LIN {X 0,Y 411.207,Z 161.266,A -85,B 0,C 180,E1 -10595.783,E2 -10595.783} C_VEL
LIN {X 0,Y 411.182,Z 161.265,A -85,B 0,C 180,E1 -10598.965,E2 -10598.965} C_VEL
LIN {X 0,Y 411.239,Z 161.26,A -85,B 0,C 180,E1 -10602.084,E2 -10602.084} C_VEL
LIN {X 0,Y 411.248,Z 161.259,A -85,B 0,C 180,E1 -10605.147,E2 -10605.147} C_VEL
LIN {X 0,Y 411.282,Z 161.252,A -85,B 0,C 180,E1 -10608.167,E2 -10608.167} C_VEL
LIN {X 0,Y 411.428,Z 161.234,A -85,B 0,C 180,E1 -10612.185,E2 -10612.185} C_VEL
LIN {X 0,Y 411.463,Z 161.231,A -85,B 0,C 180,E1 -10614.118,E2 -10614.118} C_VEL
LIN {X 0,Y 411.499,Z 161.226,A -85,B 0,C 180,E1 -10618.042,E2 -10618.042} C_VEL
LIN {X 0,Y 411.626,Z 161.21,A -85,B 0,C 180,E1 -10620,E2 -10620} C_VEL
LIN {X 0,Y 411.439,Z 161.237,A -85,B 0,C 180,E1 -10622.937,E2 -10622.937} C_VEL
LIN {X 0,Y 411.445,Z 161.234,A -85,B 0,C 180,E1 -10626.867,E2 -10626.867} C_VEL
LIN {X 0,Y 411.294,Z 161.252,A -85,B 0,C 180,E1 -10629.839,E2 -10629.839} C_VEL
LIN {X 0,Y 411.299,Z 161.251,A -85,B 0,C 180,E1 -10633.11,E2 -10633.11} C_VEL
LIN {X 0,Y 411.243,Z 161.258,A -85,B 0,C 180,E1 -10636.889,E2 -10636.889} C_VEL
LIN {X 0,Y 411.241,Z 161.261,A -85,B 0,C 180,E1 -10639.986,E2 -10639.986} C_VEL
LIN {X 0,Y 411.192,Z 161.264,A -85,B 0,C 180,E1 -10643.148,E2 -10643.148} C_VEL
LIN {X 0,Y 411.182,Z 161.268,A -85,B 0,C 180,E1 -10646.385,E2 -10646.385} C_VEL
LIN {X 0,Y 411.185,Z 161.268,A -85,B 0,C 180,E1 -10649.714,E2 -10649.714} C_VEL
LIN {X 0,Y 411.194,Z 161.265,A -85,B 0,C 180,E1 -10653.157,E2 -10653.157} C_VEL
LIN {X 0,Y 411.184,Z 161.265,A -85,B 0,C 180,E1 -10656.554,E2 -10656.554} C_VEL
LIN {X 0,Y 411.207,Z 161.266,A -85,B 0,C 180,E1 -10659.73,E2 -10659.73} C_VEL
LIN {X 0,Y 411.167,Z 161.269,A -85,B 0,C 180,E1 -10663.134,E2 -10663.134} C_VEL
LIN {X 0,Y 411.164,Z 161.27,A -85,B 0,C 180,E1 -10665.882,E2 -10665.882} C_VEL
LIN {X 0,Y 411.155,Z 161.27,A -85,B 0,C 180,E1 -10668.773,E2 -10668.773} C_VEL
LIN {X 0,Y 411.183,Z 161.264,A -85,B 0,C 180,E1 -10672.028,E2 -10672.028} C_VEL
LIN {X 0,Y 411.198,Z 161.264,A -85,B 0,C 180,E1 -10675.668,E2 -10675.668} C_VEL
LIN {X 0,Y 411.194,Z 161.266,A -85,B 0,C 180,E1 -10679.155,E2 -10679.155} C_VEL
LIN {X 0,Y 411.254,Z 161.257,A -85,B 0,C 180,E1 -10682.524,E2 -10682.524} C_VEL
LIN {X 0,Y 411.212,Z 161.26,A -85,B 0,C 180,E1 -10685.786,E2 -10685.786} C_VEL
LIN {X 0,Y 411.193,Z 161.265,A -85,B 0,C 180,E1 -10688.968,E2 -10688.968} C_VEL
LIN {X 0,Y 411.251,Z 161.259,A -85,B 0,C 180,E1 -10692.087,E2 -10692.087} C_VEL
LIN {X 0,Y 411.257,Z 161.257,A -85,B 0,C 180,E1 -10695.149,E2 -10695.149} C_VEL
LIN {X 0,Y 411.282,Z 161.255,A -85,B 0,C 180,E1 -10698.169,E2 -10698.169} C_VEL
LIN {X 0,Y 411.482,Z 161.231,A -85,B 0,C 180,E1 -10702.148,E2 -10702.148} C_VEL
LIN {X 0,Y 411.476,Z 161.231,A -85,B 0,C 180,E1 -10704.12,E2 -10704.12} C_VEL
LIN {X 0,Y 411.512,Z 161.227,A -85,B 0,C 180,E1 -10708.044,E2 -10708.044} C_VEL
LIN {X 0,Y 411.379,Z 161.239,A -85,B 0,C 180,E1 -10710.98,E2 -10710.98} C_VEL
LIN {X 0,Y 411.452,Z 161.231,A -85,B 0,C 180,E1 -10712.939,E2 -10712.939} C_VEL
LIN {X 0,Y 411.464,Z 161.231,A -85,B 0,C 180,E1 -10716.868,E2 -10716.868} C_VEL
LIN {X 0,Y 411.357,Z 161.244,A -85,B 0,C 180,E1 -10718.847,E2 -10718.847} C_VEL
LIN {X 0,Y 411.287,Z 161.255,A -85,B 0,C 180,E1 -10721.834,E2 -10721.834} C_VEL
LIN {X 0,Y 411.26,Z 161.255,A -85,B 0,C 180,E1 -10724.854,E2 -10724.854} C_VEL
LIN {X 0,Y 411.243,Z 161.258,A -85,B 0,C 180,E1 -10727.609,E2 -10727.609} C_VEL
LIN {X 0,Y 410.583,Z 161.342,A -85,B 0,C 180,E1 -10728.427,E2 -10728.427} C_VEL
LIN {X 0,Y 407.695,Z 161.704,A -85,B 0,C 180,E1 -10729.755,E2 -10729.755} C_VEL
LIN {X 0,Y 405.251,Z 162.006,A -85,B 0,C 180,E1 -10730.827,E2 -10730.827} C_VEL
LIN {X 0,Y 404.215,Z 162.136,A -85,B 0,C 180,E1 -10731.657,E2 -10731.657} C_VEL
LIN {X 0,Y 404.138,Z 162.142,A -85,B 0,C 180,E1 -10731.938,E2 -10731.938} C_VEL
LIN {X 0,Y 404.156,Z 162.144,A -85,B 0,C 180,E1 -10735.278,E2 -10735.278} C_VEL
LIN {X 0,Y 404.156,Z 162.143,A -85,B 0,C 180,E1 -10739.139,E2 -10739.139} C_VEL
LIN {X 0,Y 404.146,Z 162.144,A -85,B 0,C 180,E1 -10742.623,E2 -10742.623} C_VEL
LIN {X 0,Y 404.184,Z 162.14,A -85,B 0,C 180,E1 -10745.19,E2 -10745.19} C_VEL
LIN {X 0,Y 404.137,Z 162.147,A -85,B 0,C 180,E1 -10748.76,E2 -10748.76} C_VEL
LIN {X 0,Y 404.113,Z 162.145,A -85,B 0,C 180,E1 -10751.598,E2 -10751.598} C_VEL
LIN {X 0,Y 404.149,Z 162.143,A -85,B 0,C 180,E1 -10754.523,E2 -10754.523} C_VEL
LIN {X 0,Y 404.142,Z 162.142,A -85,B 0,C 180,E1 -10757.296,E2 -10757.296} C_VEL
LIN {X 0,Y 404.137,Z 162.144,A -85,B 0,C 180,E1 -10759.952,E2 -10759.952} C_VEL
LIN {X 0,Y 404.137,Z 162.142,A -85,B 0,C 180,E1 -10763.127,E2 -10763.127} C_VEL
LIN {X 0,Y 404.212,Z 162.136,A -85,B 0,C 180,E1 -10766.573,E2 -10766.573} C_VEL
LIN {X 0,Y 404.224,Z 162.166,A -85,B 0,C 180,E1 -10766.845,E2 -10766.845} C_VEL
LIN {X 0,Y 405.07,Z 167.315,A -85,B 0,C 180,E1 -10769.214,E2 -10769.214} C_VEL
LIN {X 0,Y 404.937,Z 172.513,A -85,B 0,C 180,E1 -10771.492,E2 -10771.492} C_VEL
LIN {X 0,Y 404.575,Z 179.708,A -85,B 0,C 180,E1 -10774.599,E2 -10774.599} C_VEL
LIN {X 0,Y 404.159,Z 187.845,A -85,B 0,C 180,E1 -10778.046,E2 -10778.046} C_VEL
LIN {X 0,Y 403.86,Z 195.462,A -85,B 0,C 180,E1 -10781.22,E2 -10781.22} C_VEL
LIN {X 0,Y 403.622,Z 203.044,A -85,B 0,C 180,E1 -10784.342,E2 -10784.342} C_VEL
LIN {X 0,Y 403.35,Z 211.861,A -85,B 0,C 180,E1 -10787.931,E2 -10787.931} C_VEL
LIN {X 0,Y 403.222,Z 215.611,A -85,B 0,C 180,E1 -10789.423,E2 -10789.423} C_VEL
LIN {X 0,Y 404.314,Z 226.159,A -85,B 0,C 180,E1 -10789.99,E2 -10789.99} C_VEL
LIN {X 0,Y 404.795,Z 233.544,A -85,B 0,C 180,E1 -10790.506,E2 -10790.506} C_VEL
LIN {X 0,Y 404.342,Z 243.511,A -85,B 0,C 180,E1 -10791.378,E2 -10791.378} C_VEL
LIN {X 0,Y 404.028,Z 251.821,A -85,B 0,C 180,E1 -10792.322,E2 -10792.322} C_VEL
LIN {X 0,Y 403.71,Z 259.93,A -85,B 0,C 180,E1 -10793.503,E2 -10793.503} C_VEL
LIN {X 0,Y 403.453,Z 266.509,A -85,B 0,C 180,E1 -10794.753,E2 -10794.753} C_VEL
LIN {X 0,Y 403.306,Z 271.492,A -85,B 0,C 180,E1 -10796.003,E2 -10796.003} C_VEL
LIN {X 0,Y 403.07,Z 275.759,A -85,B 0,C 180,E1 -10797.502,E2 -10797.502} C_VEL
LIN {X 0,Y 402.968,Z 278.356,A -85,B 0,C 180,E1 -10799.001,E2 -10799.001} C_VEL
LIN {X 0,Y 402.972,Z 279.231,A -85,B 0,C 180,E1 -10800,E2 -10800} C_VEL
LIN {X 0,Y 403.052,Z 279.432,A -85,B 0,C 180,E1 -10800.999,E2 -10800.999} C_VEL
LIN {X 0,Y 403.192,Z 278.964,A -85,B 0,C 180,E1 -10801.998,E2 -10801.998} C_VEL
LIN {X 0,Y 403.41,Z 277.828,A -85,B 0,C 180,E1 -10802.996,E2 -10802.996} C_VEL
LIN {X 0,Y 403.747,Z 274.846,A -85,B 0,C 180,E1 -10804.493,E2 -10804.493} C_VEL
LIN {X 0,Y 404.065,Z 270.202,A -85,B 0,C 180,E1 -10805.99,E2 -10805.99} C_VEL
LIN {X 0,Y 404.434,Z 264.853,A -85,B 0,C 180,E1 -10807.238,E2 -10807.238} C_VEL
LIN {X 0,Y 405.159,Z 257.556,A -85,B 0,C 180,E1 -10808.529,E2 -10808.529} C_VEL
LIN {X 0,Y 405.943,Z 248.74,A -85,B 0,C 180,E1 -10809.718,E2 -10809.718} C_VEL
LIN {X 0,Y 406.748,Z 239.232,A -85,B 0,C 180,E1 -10810.705,E2 -10810.705} C_VEL
LIN {X 0,Y 406.752,Z 233.542,A -85,B 0,C 180,E1 -10811.209,E2 -10811.209} C_VEL
LIN {X 0,Y 405.297,Z 223.531,A -85,B 0,C 180,E1 -10812.01,E2 -10812.01} C_VEL
LIN {X 0,Y 403.844,Z 216.665,A -85,B 0,C 180,E1 -10812.507,E2 -10812.507} C_VEL
LIN {X 0,Y 404.246,Z 209.533,A -85,B 0,C 180,E1 -10815.633,E2 -10815.633} C_VEL
LIN {X 0,Y 404.678,Z 202.657,A -85,B 0,C 180,E1 -10818.741,E2 -10818.741} C_VEL
LIN {X 0,Y 405.281,Z 194.834,A -85,B 0,C 180,E1 -10822.427,E2 -10822.427} C_VEL
LIN {X 0,Y 406.002,Z 188.022,A -85,B 0,C 180,E1 -10825.822,E2 -10825.822} C_VEL
LIN {X 0,Y 406.894,Z 182.208,A -85,B 0,C 180,E1 -10828.923,E2 -10828.923} C_VEL
LIN {X 0,Y 407.201,Z 178.392,A -85,B 0,C 180,E1 -10831.184,E2 -10831.184} C_VEL
LIN {X 0,Y 406.895,Z 175.006,A -85,B 0,C 180,E1 -10833.554,E2 -10833.554} C_VEL
LIN {X 0,Y 406.335,Z 172.065,A -85,B 0,C 180,E1 -10836.02,E2 -10836.02} C_VEL
LIN {X 0,Y 405.886,Z 169.428,A -85,B 0,C 180,E1 -10838.812,E2 -10838.812} C_VEL
LIN {X 0,Y 405.452,Z 167.68,A -85,B 0,C 180,E1 -10841.809,E2 -10841.809} C_VEL
LIN {X 0,Y 405.365,Z 167.011,A -85,B 0,C 180,E1 -10844.696,E2 -10844.696} C_VEL
LIN {X 0,Y 405.483,Z 167.548,A -85,B 0,C 180,E1 -10847.469,E2 -10847.469} C_VEL
LIN {X 0,Y 405.882,Z 169.048,A -85,B 0,C 180,E1 -10850.157,E2 -10850.157} C_VEL
LIN {X 0,Y 406.461,Z 171.553,A -85,B 0,C 180,E1 -10852.757,E2 -10852.757} C_VEL
LIN {X 0,Y 407.472,Z 175.865,A -85,B 0,C 180,E1 -10855.884,E2 -10855.884} C_VEL
LIN {X 0,Y 408.63,Z 181.39,A -85,B 0,C 180,E1 -10858.936,E2 -10858.936} C_VEL
LIN {X 0,Y 409.421,Z 186.484,A -85,B 0,C 180,E1 -10861.271,E2 -10861.271} C_VEL
LIN {X 0,Y 408.85,Z 190.802,A -85,B 0,C 180,E1 -10862.9,E2 -10862.9} C_VEL
LIN {X 0,Y 407.122,Z 200.495,A -85,B 0,C 180,E1 -10866.195,E2 -10866.195} C_VEL
LIN {X 0,Y 405.713,Z 211.784,A -85,B 0,C 180,E1 -10869.728,E2 -10869.728} C_VEL
LIN {X 0,Y 404.899,Z 220.511,A -85,B 0,C 180,E1 -10872.295,E2 -10872.295} C_VEL
LIN {X 0,Y 407.213,Z 233.303,A -85,B 0,C 180,E1 -10872.87,E2 -10872.87} C_VEL
LIN {X 0,Y 407.871,Z 244.837,A -85,B 0,C 180,E1 -10873.481,E2 -10873.481} C_VEL
LIN {X 0,Y 407.187,Z 256.391,A -85,B 0,C 180,E1 -10874.225,E2 -10874.225} C_VEL
LIN {X 0,Y 406.24,Z 268.36,A -85,B 0,C 180,E1 -10875.215,E2 -10875.215} C_VEL
LIN {X 0,Y 405.341,Z 278.907,A -85,B 0,C 180,E1 -10876.327,E2 -10876.327} C_VEL
LIN {X 0,Y 404.683,Z 289.375,A -85,B 0,C 180,E1 -10877.715,E2 -10877.715} C_VEL
LIN {X 0,Y 403.867,Z 298.395,A -85,B 0,C 180,E1 -10879.217,E2 -10879.217} C_VEL
LIN {X 0,Y 403.427,Z 305.665,A -85,B 0,C 180,E1 -10880.725,E2 -10880.725} C_VEL
LIN {X 0,Y 403.192,Z 310.558,A -85,B 0,C 180,E1 -10881.983,E2 -10881.983} C_VEL
LIN {X 0,Y 403.004,Z 315.426,A -85,B 0,C 180,E1 -10883.54,E2 -10883.54} C_VEL
LIN {X 0,Y 402.961,Z 318.87,A -85,B 0,C 180,E1 -10884.996,E2 -10884.996} C_VEL
LIN {X 0,Y 402.885,Z 320.644,A -85,B 0,C 180,E1 -10885.997,E2 -10885.997} C_VEL
LIN {X 0,Y 402.918,Z 322.001,A -85,B 0,C 180,E1 -10886.999,E2 -10886.999} C_VEL
LIN {X 0,Y 402.969,Z 322.941,A -85,B 0,C 180,E1 -10888,E2 -10888} C_VEL
LIN {X 0,Y 402.929,Z 323.408,A -85,B 0,C 180,E1 -10888.999,E2 -10888.999} C_VEL
LIN {X 0,Y 402.958,Z 323.469,A -85,B 0,C 180,E1 -10889.998,E2 -10889.998} C_VEL
LIN {X 0,Y 402.962,Z 323.121,A -85,B 0,C 180,E1 -10890.998,E2 -10890.998} C_VEL
LIN {X 0,Y 402.989,Z 322.303,A -85,B 0,C 180,E1 -10891.997,E2 -10891.997} C_VEL
LIN {X 0,Y 403.004,Z 321.057,A -85,B 0,C 180,E1 -10892.997,E2 -10892.997} C_VEL
LIN {X 0,Y 402.95,Z 318.326,A -85,B 0,C 180,E1 -10894.5,E2 -10894.5} C_VEL
LIN {X 0,Y 402.986,Z 314.496,A -85,B 0,C 180,E1 -10896.005,E2 -10896.005} C_VEL
LIN {X 0,Y 403.126,Z 309.461,A -85,B 0,C 180,E1 -10897.511,E2 -10897.511} C_VEL
LIN {X 0,Y 403.313,Z 302.989,A -85,B 0,C 180,E1 -10899.021,E2 -10899.021} C_VEL
LIN {X 0,Y 403.674,Z 294.844,A -85,B 0,C 180,E1 -10900.531,E2 -10900.531} C_VEL
LIN {X 0,Y 404.185,Z 286.47,A -85,B 0,C 180,E1 -10901.787,E2 -10901.787} C_VEL
LIN {X 0,Y 404.704,Z 277.19,A -85,B 0,C 180,E1 -10902.918,E2 -10902.918} C_VEL
LIN {X 0,Y 405.199,Z 265.616,A -85,B 0,C 180,E1 -10904.051,E2 -10904.051} C_VEL
LIN {X 0,Y 405.85,Z 254.099,A -85,B 0,C 180,E1 -10904.925,E2 -10904.925} C_VEL
LIN {X 0,Y 406.283,Z 242.176,A -85,B 0,C 180,E1 -10905.615,E2 -10905.615} C_VEL
LIN {X 0,Y 405.168,Z 230.504,A -85,B 0,C 180,E1 -10906.139,E2 -10906.139} C_VEL
LIN {X 0,Y 404.151,Z 220.278,A -85,B 0,C 180,E1 -10906.49,E2 -10906.49} C_VEL
LIN {X 0,Y 405.068,Z 206.335,A -85,B 0,C 180,E1 -10910.302,E2 -10910.302} C_VEL
LIN {X 0,Y 406.165,Z 193.07,A -85,B 0,C 180,E1 -10913.991,E2 -10913.991} C_VEL
LIN {X 0,Y 407.256,Z 181.733,A -85,B 0,C 180,E1 -10917.211,E2 -10917.211} C_VEL
LIN {X 0,Y 407.239,Z 177.881,A -85,B 0,C 180,E1 -10918.34,E2 -10918.34} C_VEL
LIN {X 0,Y 405.33,Z 168.24,A -85,B 0,C 180,E1 -10921.341,E2 -10921.341} C_VEL
LIN {X 0,Y 404.145,Z 162.145,A -85,B 0,C 180,E1 -10923.327,E2 -10923.327} C_VEL
LIN {X 0,Y 404.137,Z 162.147,A -85,B 0,C 180,E1 -10926.244,E2 -10926.244} C_VEL
LIN {X 0,Y 404.143,Z 162.145,A -85,B 0,C 180,E1 -10928.756,E2 -10928.756} C_VEL
LIN {X 0,Y 404.11,Z 162.144,A -85,B 0,C 180,E1 -10931.597,E2 -10931.597} C_VEL
LIN {X 0,Y 404.144,Z 162.145,A -85,B 0,C 180,E1 -10934.522,E2 -10934.522} C_VEL
LIN {X 0,Y 404.201,Z 162.135,A -85,B 0,C 180,E1 -10937.304,E2 -10937.304} C_VEL
LIN {X 0,Y 404.159,Z 162.142,A -85,B 0,C 180,E1 -10939.954,E2 -10939.954} C_VEL
LIN {X 0,Y 404.126,Z 162.143,A -85,B 0,C 180,E1 -10943.124,E2 -10943.124} C_VEL
LIN {X 0,Y 404.133,Z 162.146,A -85,B 0,C 180,E1 -10946.186,E2 -10946.186} C_VEL
LIN {X 0,Y 404.142,Z 162.146,A -85,B 0,C 180,E1 -10949.714,E2 -10949.714} C_VEL
LIN {X 0,Y 404.182,Z 162.138,A -85,B 0,C 180,E1 -10953.122,E2 -10953.122} C_VEL
LIN {X 0,Y 404.161,Z 162.14,A -85,B 0,C 180,E1 -10955.333,E2 -10955.333} C_VEL
LIN {X 0,Y 404.124,Z 162.144,A -85,B 0,C 180,E1 -10958.58,E2 -10958.58} C_VEL
LIN {X 0,Y 404.196,Z 162.137,A -85,B 0,C 180,E1 -10961.761,E2 -10961.761} C_VEL
LIN {X 0,Y 404.193,Z 162.137,A -85,B 0,C 180,E1 -10964.881,E2 -10964.881} C_VEL
LIN {X 0,Y 404.253,Z 162.129,A -85,B 0,C 180,E1 -10967.958,E2 -10967.958} C_VEL
LIN {X 0,Y 404.391,Z 162.111,A -85,B 0,C 180,E1 -10972.127,E2 -10972.127} C_VEL
LIN {X 0,Y 404.411,Z 162.109,A -85,B 0,C 180,E1 -10974.015,E2 -10974.015} C_VEL
LIN {X 0,Y 404.468,Z 162.102,A -85,B 0,C 180,E1 -10978.008,E2 -10978.008} C_VEL
LIN {X 0,Y 404.595,Z 162.085,A -85,B 0,C 180,E1 -10980,E2 -10980} C_VEL
LIN {X 0,Y 404.397,Z 162.114,A -85,B 0,C 180,E1 -10982.989,E2 -10982.989} C_VEL
LIN {X 0,Y 404.396,Z 162.112,A -85,B 0,C 180,E1 -10986.987,E2 -10986.987} C_VEL
LIN {X 0,Y 404.257,Z 162.129,A -85,B 0,C 180,E1 -10990.012,E2 -10990.012} C_VEL
LIN {X 0,Y 404.252,Z 162.128,A -85,B 0,C 180,E1 -10993.212,E2 -10993.212} C_VEL
LIN {X 0,Y 404.201,Z 162.135,A -85,B 0,C 180,E1 -10997.008,E2 -10997.008} C_VEL
LIN {X 0,Y 404.187,Z 162.139,A -85,B 0,C 180,E1 -11000.35,E2 -11000.35} C_VEL
LIN {X 0,Y 404.155,Z 162.142,A -85,B 0,C 180,E1 -11003.575,E2 -11003.575} C_VEL
LIN {X 0,Y 404.121,Z 162.144,A -85,B 0,C 180,E1 -11006.882,E2 -11006.882} C_VEL
LIN {X 0,Y 404.131,Z 162.145,A -85,B 0,C 180,E1 -11010.286,E2 -11010.286} C_VEL
LIN {X 0,Y 404.133,Z 162.146,A -85,B 0,C 180,E1 -11013.813,E2 -11013.813} C_VEL
LIN {X 0,Y 404.128,Z 162.144,A -85,B 0,C 180,E1 -11016.877,E2 -11016.877} C_VEL
LIN {X 0,Y 404.137,Z 162.143,A -85,B 0,C 180,E1 -11020.082,E2 -11020.082} C_VEL
LIN {X 0,Y 404.146,Z 162.143,A -85,B 0,C 180,E1 -11023.086,E2 -11023.086} C_VEL
LIN {X 0,Y 404.143,Z 162.144,A -85,B 0,C 180,E1 -11025.928,E2 -11025.928} C_VEL
LIN {X 0,Y 404.11,Z 162.147,A -85,B 0,C 180,E1 -11028.637,E2 -11028.637} C_VEL
LIN {X 0,Y 404.141,Z 162.145,A -85,B 0,C 180,E1 -11031.495,E2 -11031.495} C_VEL
LIN {X 0,Y 404.177,Z 162.142,A -85,B 0,C 180,E1 -11034.986,E2 -11034.986} C_VEL
LIN {X 0,Y 404.141,Z 162.144,A -85,B 0,C 180,E1 -11038.556,E2 -11038.556} C_VEL
LIN {X 0,Y 404.192,Z 162.136,A -85,B 0,C 180,E1 -11042.002,E2 -11042.002} C_VEL
LIN {X 0,Y 404.168,Z 162.139,A -85,B 0,C 180,E1 -11045.336,E2 -11045.336} C_VEL
LIN {X 0,Y 404.156,Z 162.144,A -85,B 0,C 180,E1 -11048.584,E2 -11048.584} C_VEL
LIN {X 0,Y 404.208,Z 162.134,A -85,B 0,C 180,E1 -11051.764,E2 -11051.764} C_VEL
LIN {X 0,Y 404.203,Z 162.137,A -85,B 0,C 180,E1 -11054.884,E2 -11054.884} C_VEL
LIN {X 0,Y 404.254,Z 162.129,A -85,B 0,C 180,E1 -11057.96,E2 -11057.96} C_VEL
LIN {X 0,Y 404.434,Z 162.109,A -85,B 0,C 180,E1 -11062.101,E2 -11062.101} C_VEL
LIN {X 0,Y 404.425,Z 162.11,A -85,B 0,C 180,E1 -11064.017,E2 -11064.017} C_VEL
LIN {X 0,Y 404.481,Z 162.102,A -85,B 0,C 180,E1 -11068.01,E2 -11068.01} C_VEL
LIN {X 0,Y 404.349,Z 162.115,A -85,B 0,C 180,E1 -11070.997,E2 -11070.997} C_VEL
LIN {X 0,Y 404.41,Z 162.108,A -85,B 0,C 180,E1 -11072.99,E2 -11072.99} C_VEL
LIN {X 0,Y 404.415,Z 162.109,A -85,B 0,C 180,E1 -11076.989,E2 -11076.989} C_VEL
LIN {X 0,Y 404.26,Z 162.13,A -85,B 0,C 180,E1 -11080.013,E2 -11080.013} C_VEL
LIN {X 0,Y 404.27,Z 162.127,A -85,B 0,C 180,E1 -11083.213,E2 -11083.213} C_VEL
LIN {X 0,Y 404.22,Z 162.135,A -85,B 0,C 180,E1 -11087.008,E2 -11087.008} C_VEL
LIN {X 0,Y 404.168,Z 162.139,A -85,B 0,C 180,E1 -11090.353,E2 -11090.353} C_VEL
LIN {X 0,Y 404.138,Z 162.142,A -85,B 0,C 180,E1 -11091.938,E2 -11091.938} C_VEL
LIN {X 0,Y 403.497,Z 162.224,A -85,B 0,C 180,E1 -11092.77,E2 -11092.77} C_VEL
LIN {X 0,Y 400.665,Z 162.576,A -85,B 0,C 180,E1 -11094.121,E2 -11094.121} C_VEL
LIN {X 0,Y 398.238,Z 162.882,A -85,B 0,C 180,E1 -11095.213,E2 -11095.213} C_VEL
LIN {X 0,Y 397.173,Z 163.01,A -85,B 0,C 180,E1 -11096.056,E2 -11096.056} C_VEL
LIN {X 0,Y 397.074,Z 163.02,A -85,B 0,C 180,E1 -11096.342,E2 -11096.342} C_VEL
LIN {X 0,Y 397.104,Z 163.019,A -85,B 0,C 180,E1 -11099.864,E2 -11099.864} C_VEL
LIN {X 0,Y 397.123,Z 163.017,A -85,B 0,C 180,E1 -11103.719,E2 -11103.719} C_VEL
LIN {X 0,Y 397.093,Z 163.021,A -85,B 0,C 180,E1 -11107.209,E2 -11107.209} C_VEL
LIN {X 0,Y 397.06,Z 163.027,A -85,B 0,C 180,E1 -11110.438,E2 -11110.438} C_VEL
LIN {X 0,Y 397.103,Z 163.019,A -85,B 0,C 180,E1 -11113.65,E2 -11113.65} C_VEL
LIN {X 0,Y 397.107,Z 163.021,A -85,B 0,C 180,E1 -11116.522,E2 -11116.522} C_VEL
LIN {X 0,Y 397.107,Z 163.018,A -85,B 0,C 180,E1 -11119.555,E2 -11119.555} C_VEL
LIN {X 0,Y 397.099,Z 163.019,A -85,B 0,C 180,E1 -11123.005,E2 -11123.005} C_VEL
LIN {X 0,Y 397.179,Z 163.072,A -85,B 0,C 180,E1 -11126.733,E2 -11126.733} C_VEL
LIN {X 0,Y 398.056,Z 168.37,A -85,B 0,C 180,E1 -11129.202,E2 -11129.202} C_VEL
LIN {X 0,Y 397.847,Z 174.757,A -85,B 0,C 180,E1 -11132.039,E2 -11132.039} C_VEL
LIN {X 0,Y 397.474,Z 181.305,A -85,B 0,C 180,E1 -11134.89,E2 -11134.89} C_VEL
LIN {X 0,Y 397.066,Z 190.251,A -85,B 0,C 180,E1 -11138.725,E2 -11138.725} C_VEL
LIN {X 0,Y 396.694,Z 199.128,A -85,B 0,C 180,E1 -11142.472,E2 -11142.472} C_VEL
LIN {X 0,Y 396.395,Z 207.989,A -85,B 0,C 180,E1 -11146.152,E2 -11146.152} C_VEL
LIN {X 0,Y 396.182,Z 215.595,A -85,B 0,C 180,E1 -11149.265,E2 -11149.265} C_VEL
LIN {X 0,Y 397.347,Z 227.437,A -85,B 0,C 180,E1 -11149.941,E2 -11149.941} C_VEL
LIN {X 0,Y 397.711,Z 234.605,A -85,B 0,C 180,E1 -11150.464,E2 -11150.464} C_VEL
LIN {X 0,Y 397.252,Z 244.375,A -85,B 0,C 180,E1 -11151.351,E2 -11151.351} C_VEL
LIN {X 0,Y 396.901,Z 253.364,A -85,B 0,C 180,E1 -11152.42,E2 -11152.42} C_VEL
LIN {X 0,Y 396.646,Z 260.068,A -85,B 0,C 180,E1 -11153.432,E2 -11153.432} C_VEL
LIN {X 0,Y 396.397,Z 266.487,A -85,B 0,C 180,E1 -11154.659,E2 -11154.659} C_VEL
LIN {X 0,Y 396.216,Z 271.57,A -85,B 0,C 180,E1 -11155.931,E2 -11155.931} C_VEL
LIN {X 0,Y 396.004,Z 275.949,A -85,B 0,C 180,E1 -11157.457,E2 -11157.457} C_VEL
LIN {X 0,Y 395.893,Z 278.654,A -85,B 0,C 180,E1 -11158.983,E2 -11158.983} C_VEL
LIN {X 0,Y 395.893,Z 279.596,A -85,B 0,C 180,E1 -11160,E2 -11160} C_VEL
LIN {X 0,Y 395.973,Z 279.868,A -85,B 0,C 180,E1 -11161.017,E2 -11161.017} C_VEL
LIN {X 0,Y 396.118,Z 279.475,A -85,B 0,C 180,E1 -11162.034,E2 -11162.034} C_VEL
LIN {X 0,Y 396.346,Z 278.414,A -85,B 0,C 180,E1 -11163.049,E2 -11163.049} C_VEL
LIN {X 0,Y 396.719,Z 275.551,A -85,B 0,C 180,E1 -11164.573,E2 -11164.573} C_VEL
LIN {X 0,Y 397.06,Z 271.053,A -85,B 0,C 180,E1 -11166.096,E2 -11166.096} C_VEL
LIN {X 0,Y 397.439,Z 266.033,A -85,B 0,C 180,E1 -11167.33,E2 -11167.33} C_VEL
LIN {X 0,Y 398.202,Z 259.079,A -85,B 0,C 180,E1 -11168.629,E2 -11168.629} C_VEL
LIN {X 0,Y 399.072,Z 250.28,A -85,B 0,C 180,E1 -11169.887,E2 -11169.887} C_VEL
LIN {X 0,Y 399.921,Z 241.18,A -85,B 0,C 180,E1 -11170.89,E2 -11170.89} C_VEL
LIN {X 0,Y 400.101,Z 235.734,A -85,B 0,C 180,E1 -11171.397,E2 -11171.397} C_VEL
LIN {X 0,Y 398.891,Z 226.392,A -85,B 0,C 180,E1 -11172.206,E2 -11172.206} C_VEL
LIN {X 0,Y 396.89,Z 216.809,A -85,B 0,C 180,E1 -11172.936,E2 -11172.936} C_VEL
LIN {X 0,Y 397.344,Z 209.011,A -85,B 0,C 180,E1 -11176.439,E2 -11176.439} C_VEL
LIN {X 0,Y 397.828,Z 202.204,A -85,B 0,C 180,E1 -11179.612,E2 -11179.612} C_VEL
LIN {X 0,Y 398.421,Z 195.601,A -85,B 0,C 180,E1 -11182.835,E2 -11182.835} C_VEL
LIN {X 0,Y 399.182,Z 189.217,A -85,B 0,C 180,E1 -11186.114,E2 -11186.114} C_VEL
LIN {X 0,Y 399.897,Z 184.831,A -85,B 0,C 180,E1 -11188.509,E2 -11188.509} C_VEL
LIN {X 0,Y 400.346,Z 181.227,A -85,B 0,C 180,E1 -11190.661,E2 -11190.661} C_VEL
LIN {X 0,Y 400.205,Z 177.886,A -85,B 0,C 180,E1 -11192.983,E2 -11192.983} C_VEL
LIN {X 0,Y 399.628,Z 174.35,A -85,B 0,C 180,E1 -11196.003,E2 -11196.003} C_VEL
LIN {X 0,Y 399.126,Z 171.446,A -85,B 0,C 180,E1 -11199.339,E2 -11199.339} C_VEL
LIN {X 0,Y 398.778,Z 169.993,A -85,B 0,C 180,E1 -11202.25,E2 -11202.25} C_VEL
LIN {X 0,Y 398.752,Z 169.62,A -85,B 0,C 180,E1 -11205.169,E2 -11205.169} C_VEL
LIN {X 0,Y 398.911,Z 170.331,A -85,B 0,C 180,E1 -11207.971,E2 -11207.971} C_VEL
LIN {X 0,Y 399.385,Z 172.082,A -85,B 0,C 180,E1 -11210.739,E2 -11210.739} C_VEL
LIN {X 0,Y 400.151,Z 175.491,A -85,B 0,C 180,E1 -11213.893,E2 -11213.893} C_VEL
LIN {X 0,Y 401.005,Z 179.27,A -85,B 0,C 180,E1 -11216.49,E2 -11216.49} C_VEL
LIN {X 0,Y 401.926,Z 183.711,A -85,B 0,C 180,E1 -11218.96,E2 -11218.96} C_VEL
LIN {X 0,Y 402.606,Z 188.858,A -85,B 0,C 180,E1 -11221.345,E2 -11221.345} C_VEL
LIN {X 0,Y 401.826,Z 193.533,A -85,B 0,C 180,E1 -11223.126,E2 -11223.126} C_VEL
LIN {X 0,Y 400.175,Z 202.295,A -85,B 0,C 180,E1 -11226.174,E2 -11226.174} C_VEL
LIN {X 0,Y 398.863,Z 212.184,A -85,B 0,C 180,E1 -11229.364,E2 -11229.364} C_VEL
LIN {X 0,Y 398.027,Z 220.376,A -85,B 0,C 180,E1 -11231.857,E2 -11231.857} C_VEL
LIN {X 0,Y 400.43,Z 233.45,A -85,B 0,C 180,E1 -11232.494,E2 -11232.494} C_VEL
LIN {X 0,Y 401.188,Z 243.95,A -85,B 0,C 180,E1 -11233.077,E2 -11233.077} C_VEL
LIN {X 0,Y 400.516,Z 255.473,A -85,B 0,C 180,E1 -11233.824,E2 -11233.824} C_VEL
LIN {X 0,Y 399.55,Z 267.51,A -85,B 0,C 180,E1 -11234.831,E2 -11234.831} C_VEL
LIN {X 0,Y 398.58,Z 277.977,A -85,B 0,C 180,E1 -11235.94,E2 -11235.94} C_VEL
LIN {X 0,Y 397.943,Z 286.02,A -85,B 0,C 180,E1 -11236.985,E2 -11236.985} C_VEL
LIN {X 0,Y 397.293,Z 294.184,A -85,B 0,C 180,E1 -11238.261,E2 -11238.261} C_VEL
LIN {X 0,Y 396.653,Z 302.202,A -85,B 0,C 180,E1 -11239.793,E2 -11239.793} C_VEL
LIN {X 0,Y 396.215,Z 308.577,A -85,B 0,C 180,E1 -11241.327,E2 -11241.327} C_VEL
LIN {X 0,Y 396.002,Z 313.635,A -85,B 0,C 180,E1 -11242.862,E2 -11242.862} C_VEL
LIN {X 0,Y 395.832,Z 317.074,A -85,B 0,C 180,E1 -11244.187,E2 -11244.187} C_VEL
LIN {X 0,Y 395.806,Z 320.34,A -85,B 0,C 180,E1 -11245.926,E2 -11245.926} C_VEL
LIN {X 0,Y 395.817,Z 321.672,A -85,B 0,C 180,E1 -11246.945,E2 -11246.945} C_VEL
LIN {X 0,Y 395.898,Z 322.567,A -85,B 0,C 180,E1 -11247.964,E2 -11247.964} C_VEL
LIN {X 0,Y 395.855,Z 323.004,A -85,B 0,C 180,E1 -11248.981,E2 -11248.981} C_VEL
LIN {X 0,Y 395.88,Z 323.039,A -85,B 0,C 180,E1 -11249.998,E2 -11249.998} C_VEL
LIN {X 0,Y 395.886,Z 322.648,A -85,B 0,C 180,E1 -11251.016,E2 -11251.016} C_VEL
LIN {X 0,Y 395.92,Z 321.791,A -85,B 0,C 180,E1 -11252.033,E2 -11252.033} C_VEL
LIN {X 0,Y 395.906,Z 320.514,A -85,B 0,C 180,E1 -11253.051,E2 -11253.051} C_VEL
LIN {X 0,Y 395.884,Z 317.722,A -85,B 0,C 180,E1 -11254.58,E2 -11254.58} C_VEL
LIN {X 0,Y 395.953,Z 313.287,A -85,B 0,C 180,E1 -11256.29,E2 -11256.29} C_VEL
LIN {X 0,Y 396.092,Z 307.669,A -85,B 0,C 180,E1 -11257.902,E2 -11257.902} C_VEL
LIN {X 0,Y 396.355,Z 300.86,A -85,B 0,C 180,E1 -11259.438,E2 -11259.438} C_VEL
LIN {X 0,Y 396.651,Z 293.835,A -85,B 0,C 180,E1 -11260.72,E2 -11260.72} C_VEL
LIN {X 0,Y 397.143,Z 285.255,A -85,B 0,C 180,E1 -11261.999,E2 -11261.999} C_VEL
LIN {X 0,Y 397.756,Z 274.619,A -85,B 0,C 180,E1 -11263.278,E2 -11263.278} C_VEL
LIN {X 0,Y 398.26,Z 263.926,A -85,B 0,C 180,E1 -11264.301,E2 -11264.301} C_VEL
LIN {X 0,Y 398.91,Z 251.981,A -85,B 0,C 180,E1 -11265.191,E2 -11265.191} C_VEL
LIN {X 0,Y 399.153,Z 240.726,A -85,B 0,C 180,E1 -11265.836,E2 -11265.836} C_VEL
LIN {X 0,Y 397.781,Z 227.494,A -85,B 0,C 180,E1 -11266.402,E2 -11266.402} C_VEL
LIN {X 0,Y 397.101,Z 220.32,A -85,B 0,C 180,E1 -11266.634,E2 -11266.634} C_VEL
LIN {X 0,Y 397.971,Z 207.811,A -85,B 0,C 180,E1 -11270.133,E2 -11270.133} C_VEL
LIN {X 0,Y 399.104,Z 194.568,A -85,B 0,C 180,E1 -11273.89,E2 -11273.89} C_VEL
LIN {X 0,Y 400.211,Z 183.208,A -85,B 0,C 180,E1 -11277.164,E2 -11277.164} C_VEL
LIN {X 0,Y 400.273,Z 179.415,A -85,B 0,C 180,E1 -11278.296,E2 -11278.296} C_VEL
LIN {X 0,Y 398.405,Z 169.781,A -85,B 0,C 180,E1 -11281.356,E2 -11281.356} C_VEL
LIN {X 0,Y 397.104,Z 163.023,A -85,B 0,C 180,E1 -11283.626,E2 -11283.626} C_VEL
LIN {X 0,Y 397.094,Z 163.023,A -85,B 0,C 180,E1 -11286.993,E2 -11286.993} C_VEL
LIN {X 0,Y 397.105,Z 163.018,A -85,B 0,C 180,E1 -11289.576,E2 -11289.576} C_VEL
LIN {X 0,Y 397.092,Z 163.019,A -85,B 0,C 180,E1 -11293.647,E2 -11293.647} C_VEL
LIN {X 0,Y 397.155,Z 163.015,A -85,B 0,C 180,E1 -11296.51,E2 -11296.51} C_VEL
LIN {X 0,Y 397.114,Z 163.018,A -85,B 0,C 180,E1 -11299.549,E2 -11299.549} C_VEL
LIN {X 0,Y 397.084,Z 163.022,A -85,B 0,C 180,E1 -11302.789,E2 -11302.789} C_VEL
LIN {X 0,Y 397.107,Z 163.021,A -85,B 0,C 180,E1 -11306.281,E2 -11306.281} C_VEL
LIN {X 0,Y 397.102,Z 163.021,A -85,B 0,C 180,E1 -11310.132,E2 -11310.132} C_VEL
LIN {X 0,Y 397.182,Z 163.01,A -85,B 0,C 180,E1 -11312.609,E2 -11312.609} C_VEL
LIN {X 0,Y 397.115,Z 163.021,A -85,B 0,C 180,E1 -11315.98,E2 -11315.98} C_VEL
LIN {X 0,Y 397.125,Z 163.019,A -85,B 0,C 180,E1 -11319.704,E2 -11319.704} C_VEL
LIN {X 0,Y 397.168,Z 163.012,A -85,B 0,C 180,E1 -11322.844,E2 -11322.844} C_VEL
LIN {X 0,Y 397.212,Z 163.005,A -85,B 0,C 180,E1 -11326.678,E2 -11326.678} C_VEL
LIN {X 0,Y 397.205,Z 163.006,A -85,B 0,C 180,E1 -11329.809,E2 -11329.809} C_VEL
LIN {X 0,Y 397.342,Z 162.992,A -85,B 0,C 180,E1 -11332.888,E2 -11332.888} C_VEL
LIN {X 0,Y 397.245,Z 163.005,A -85,B 0,C 180,E1 -11334.925,E2 -11334.925} C_VEL
LIN {X 0,Y 397.437,Z 162.977,A -85,B 0,C 180,E1 -11337.973,E2 -11337.973} C_VEL
LIN {X 0,Y 397.565,Z 162.961,A -85,B 0,C 180,E1 -11340,E2 -11340} C_VEL
LIN {X 0,Y 397.357,Z 162.99,A -85,B 0,C 180,E1 -11343.042,E2 -11343.042} C_VEL
LIN {X 0,Y 397.349,Z 162.99,A -85,B 0,C 180,E1 -11347.112,E2 -11347.112} C_VEL
LIN {X 0,Y 397.215,Z 163.007,A -85,B 0,C 180,E1 -11350.191,E2 -11350.191} C_VEL
LIN {X 0,Y 397.212,Z 163.005,A -85,B 0,C 180,E1 -11353.321,E2 -11353.321} C_VEL
LIN {X 0,Y 397.167,Z 163.011,A -85,B 0,C 180,E1 -11357.156,E2 -11357.156} C_VEL
LIN {X 0,Y 397.119,Z 163.02,A -85,B 0,C 180,E1 -11360.729,E2 -11360.729} C_VEL
LIN {X 0,Y 397.117,Z 163.019,A -85,B 0,C 180,E1 -11364.019,E2 -11364.019} C_VEL
LIN {X 0,Y 397.088,Z 163.02,A -85,B 0,C 180,E1 -11367.398,E2 -11367.398} C_VEL
LIN {X 0,Y 397.065,Z 163.023,A -85,B 0,C 180,E1 -11370.884,E2 -11370.884} C_VEL
LIN {X 0,Y 397.114,Z 163.019,A -85,B 0,C 180,E1 -11374.494,E2 -11374.494} C_VEL
LIN {X 0,Y 397.095,Z 163.02,A -85,B 0,C 180,E1 -11378.276,E2 -11378.276} C_VEL
LIN {X 0,Y 397.079,Z 163.021,A -85,B 0,C 180,E1 -11380.91,E2 -11380.91} C_VEL
LIN {X 0,Y 397.094,Z 163.022,A -85,B 0,C 180,E1 -11383.65,E2 -11383.65} C_VEL
LIN {X 0,Y 397.095,Z 163.02,A -85,B 0,C 180,E1 -11386.522,E2 -11386.522} C_VEL
LIN {X 0,Y 397.104,Z 163.018,A -85,B 0,C 180,E1 -11390.424,E2 -11390.424} C_VEL
LIN {X 0,Y 397.1,Z 163.018,A -85,B 0,C 180,E1 -11394.267,E2 -11394.267} C_VEL
LIN {X 0,Y 397.108,Z 163.021,A -85,B 0,C 180,E1 -11396.729,E2 -11396.729} C_VEL
LIN {X 0,Y 397.128,Z 163.017,A -85,B 0,C 180,E1 -11400.298,E2 -11400.298} C_VEL
LIN {X 0,Y 397.189,Z 163.01,A -85,B 0,C 180,E1 -11402.612,E2 -11402.612} C_VEL
LIN {X 0,Y 397.124,Z 163.015,A -85,B 0,C 180,E1 -11405.983,E2 -11405.983} C_VEL
LIN {X 0,Y 397.136,Z 163.015,A -85,B 0,C 180,E1 -11409.706,E2 -11409.706} C_VEL
LIN {X 0,Y 397.18,Z 163.013,A -85,B 0,C 180,E1 -11412.847,E2 -11412.847} C_VEL
LIN {X 0,Y 397.227,Z 163.006,A -85,B 0,C 180,E1 -11416.704,E2 -11416.704} C_VEL
LIN {X 0,Y 397.216,Z 163.005,A -85,B 0,C 180,E1 -11419.811,E2 -11419.811} C_VEL
LIN {X 0,Y 397.365,Z 162.987,A -85,B 0,C 180,E1 -11422.89,E2 -11422.89} C_VEL
LIN {X 0,Y 397.256,Z 163.001,A -85,B 0,C 180,E1 -11424.927,E2 -11424.927} C_VEL
LIN {X 0,Y 397.45,Z 162.978,A -85,B 0,C 180,E1 -11427.975,E2 -11427.975} C_VEL
LIN {X 0,Y 397.32,Z 162.99,A -85,B 0,C 180,E1 -11431.015,E2 -11431.015} C_VEL
LIN {X 0,Y 397.37,Z 162.985,A -85,B 0,C 180,E1 -11433.043,E2 -11433.043} C_VEL
LIN {X 0,Y 397.367,Z 162.987,A -85,B 0,C 180,E1 -11437.113,E2 -11437.113} C_VEL
LIN {X 0,Y 397.22,Z 163.005,A -85,B 0,C 180,E1 -11440.192,E2 -11440.192} C_VEL
LIN {X 0,Y 397.23,Z 163.005,A -85,B 0,C 180,E1 -11443.322,E2 -11443.322} C_VEL
LIN {X 0,Y 397.186,Z 163.012,A -85,B 0,C 180,E1 -11447.156,E2 -11447.156} C_VEL
LIN {X 0,Y 397.107,Z 163.02,A -85,B 0,C 180,E1 -11450.731,E2 -11450.731} C_VEL
LIN {X 0,Y 397.111,Z 163.017,A -85,B 0,C 180,E1 -11454.021,E2 -11454.021} C_VEL
LIN {X 0,Y 397.074,Z 163.02,A -85,B 0,C 180,E1 -11456.342,E2 -11456.342} C_VEL
LIN {X 0,Y 396.378,Z 163.112,A -85,B 0,C 180,E1 -11457.189,E2 -11457.189} C_VEL
LIN {X 0,Y 393.526,Z 163.466,A -85,B 0,C 180,E1 -11458.566,E2 -11458.566} C_VEL
LIN {X 0,Y 391.129,Z 163.764,A -85,B 0,C 180,E1 -11459.678,E2 -11459.678} C_VEL
LIN {X 0,Y 390.1,Z 163.893,A -85,B 0,C 180,E1 -11460.538,E2 -11460.538} C_VEL
LIN {X 0,Y 390.014,Z 163.9,A -85,B 0,C 180,E1 -11460.829,E2 -11460.829} C_VEL
LIN {X 0,Y 390.073,Z 163.895,A -85,B 0,C 180,E1 -11464.026,E2 -11464.026} C_VEL
LIN {X 0,Y 390.042,Z 163.897,A -85,B 0,C 180,E1 -11467.55,E2 -11467.55} C_VEL
LIN {X 0,Y 390.022,Z 163.903,A -85,B 0,C 180,E1 -11470.815,E2 -11470.815} C_VEL
LIN {X 0,Y 390.057,Z 163.897,A -85,B 0,C 180,E1 -11473.886,E2 -11473.886} C_VEL
LIN {X 0,Y 390.062,Z 163.899,A -85,B 0,C 180,E1 -11476.79,E2 -11476.79} C_VEL
LIN {X 0,Y 390.061,Z 163.896,A -85,B 0,C 180,E1 -11479.561,E2 -11479.561} C_VEL
LIN {X 0,Y 390.044,Z 163.9,A -85,B 0,C 180,E1 -11482.451,E2 -11482.451} C_VEL
LIN {X 0,Y 390.107,Z 163.893,A -85,B 0,C 180,E1 -11486.049,E2 -11486.049} C_VEL
LIN {X 0,Y 390.17,Z 164.088,A -85,B 0,C 180,E1 -11486.675,E2 -11486.675} C_VEL
LIN {X 0,Y 391.018,Z 169.32,A -85,B 0,C 180,E1 -11489.152,E2 -11489.152} C_VEL
LIN {X 0,Y 390.832,Z 175.164,A -85,B 0,C 180,E1 -11491.78,E2 -11491.78} C_VEL
LIN {X 0,Y 390.416,Z 182.374,A -85,B 0,C 180,E1 -11494.974,E2 -11494.974} C_VEL
LIN {X 0,Y 389.969,Z 191.344,A -85,B 0,C 180,E1 -11498.873,E2 -11498.873} C_VEL
LIN {X 0,Y 389.666,Z 198.998,A -85,B 0,C 180,E1 -11502.145,E2 -11502.145} C_VEL
LIN {X 0,Y 389.343,Z 207.885,A -85,B 0,C 180,E1 -11505.896,E2 -11505.896} C_VEL
LIN {X 0,Y 389.12,Z 215.655,A -85,B 0,C 180,E1 -11509.134,E2 -11509.134} C_VEL
LIN {X 0,Y 390.261,Z 227.593,A -85,B 0,C 180,E1 -11509.822,E2 -11509.822} C_VEL
LIN {X 0,Y 390.694,Z 233.942,A -85,B 0,C 180,E1 -11510.291,E2 -11510.291} C_VEL
LIN {X 0,Y 390.237,Z 243.888,A -85,B 0,C 180,E1 -11511.195,E2 -11511.195} C_VEL
LIN {X 0,Y 389.851,Z 253.062,A -85,B 0,C 180,E1 -11512.282,E2 -11512.282} C_VEL
LIN {X 0,Y 389.576,Z 260.296,A -85,B 0,C 180,E1 -11513.381,E2 -11513.381} C_VEL
LIN {X 0,Y 389.345,Z 266.434,A -85,B 0,C 180,E1 -11514.562,E2 -11514.562} C_VEL
LIN {X 0,Y 389.127,Z 271.629,A -85,B 0,C 180,E1 -11515.857,E2 -11515.857} C_VEL
LIN {X 0,Y 388.938,Z 276.116,A -85,B 0,C 180,E1 -11517.411,E2 -11517.411} C_VEL
LIN {X 0,Y 388.82,Z 278.935,A -85,B 0,C 180,E1 -11518.964,E2 -11518.964} C_VEL
LIN {X 0,Y 388.817,Z 279.955,A -85,B 0,C 180,E1 -11520,E2 -11520} C_VEL
LIN {X 0,Y 388.898,Z 280.306,A -85,B 0,C 180,E1 -11521.036,E2 -11521.036} C_VEL
LIN {X 0,Y 389.048,Z 279.992,A -85,B 0,C 180,E1 -11522.071,E2 -11522.071} C_VEL
LIN {X 0,Y 389.285,Z 279.016,A -85,B 0,C 180,E1 -11523.105,E2 -11523.105} C_VEL
LIN {X 0,Y 389.655,Z 277.356,A -85,B 0,C 180,E1 -11524.137,E2 -11524.137} C_VEL
LIN {X 0,Y 389.865,Z 273.584,A -85,B 0,C 180,E1 -11525.69,E2 -11525.69} C_VEL
LIN {X 0,Y 390.332,Z 268.04,A -85,B 0,C 180,E1 -11527.241,E2 -11527.241} C_VEL
LIN {X 0,Y 391.079,Z 261.792,A -85,B 0,C 180,E1 -11528.526,E2 -11528.526} C_VEL
LIN {X 0,Y 392.023,Z 253.727,A -85,B 0,C 180,E1 -11529.806,E2 -11529.806} C_VEL
LIN {X 0,Y 392.836,Z 245.507,A -85,B 0,C 180,E1 -11530.827,E2 -11530.827} C_VEL
LIN {X 0,Y 393.452,Z 237.937,A -85,B 0,C 180,E1 -11531.593,E2 -11531.593} C_VEL
LIN {X 0,Y 392.312,Z 228.2,A -85,B 0,C 180,E1 -11532.495,E2 -11532.495} C_VEL
LIN {X 0,Y 389.944,Z 216.87,A -85,B 0,C 180,E1 -11533.423,E2 -11533.423} C_VEL
LIN {X 0,Y 390.392,Z 209.683,A -85,B 0,C 180,E1 -11536.741,E2 -11536.741} C_VEL
LIN {X 0,Y 390.925,Z 202.932,A -85,B 0,C 180,E1 -11539.973,E2 -11539.973} C_VEL
LIN {X 0,Y 391.567,Z 196.385,A -85,B 0,C 180,E1 -11543.258,E2 -11543.258} C_VEL
LIN {X 0,Y 392.398,Z 190.14,A -85,B 0,C 180,E1 -11546.6,E2 -11546.6} C_VEL
LIN {X 0,Y 393.123,Z 186.169,A -85,B 0,C 180,E1 -11548.861,E2 -11548.861} C_VEL
LIN {X 0,Y 393.54,Z 182.47,A -85,B 0,C 180,E1 -11551.191,E2 -11551.191} C_VEL
LIN {X 0,Y 393.451,Z 180.111,A -85,B 0,C 180,E1 -11552.907,E2 -11552.907} C_VEL
LIN {X 0,Y 392.862,Z 176.447,A -85,B 0,C 180,E1 -11556.182,E2 -11556.182} C_VEL
LIN {X 0,Y 392.496,Z 174.248,A -85,B 0,C 180,E1 -11558.808,E2 -11558.808} C_VEL
LIN {X 0,Y 392.169,Z 172.796,A -85,B 0,C 180,E1 -11561.535,E2 -11561.535} C_VEL
LIN {X 0,Y 392.121,Z 172.165,A -85,B 0,C 180,E1 -11564.347,E2 -11564.347} C_VEL
LIN {X 0,Y 392.247,Z 172.66,A -85,B 0,C 180,E1 -11567.274,E2 -11567.274} C_VEL
LIN {X 0,Y 392.693,Z 174.344,A -85,B 0,C 180,E1 -11570.316,E2 -11570.316} C_VEL
LIN {X 0,Y 393.133,Z 176.445,A -85,B 0,C 180,E1 -11572.567,E2 -11572.567} C_VEL
LIN {X 0,Y 393.897,Z 179.71,A -85,B 0,C 180,E1 -11575.182,E2 -11575.182} C_VEL
LIN {X 0,Y 394.757,Z 183.72,A -85,B 0,C 180,E1 -11577.716,E2 -11577.716} C_VEL
LIN {X 0,Y 395.599,Z 188.449,A -85,B 0,C 180,E1 -11580.168,E2 -11580.168} C_VEL
LIN {X 0,Y 395.784,Z 191.039,A -85,B 0,C 180,E1 -11581.35,E2 -11581.35} C_VEL
LIN {X 0,Y 394.685,Z 196.816,A -85,B 0,C 180,E1 -11583.565,E2 -11583.565} C_VEL
LIN {X 0,Y 392.722,Z 207.699,A -85,B 0,C 180,E1 -11587.37,E2 -11587.37} C_VEL
LIN {X 0,Y 391.271,Z 219.488,A -85,B 0,C 180,E1 -11591.135,E2 -11591.135} C_VEL
LIN {X 0,Y 391.186,Z 220.438,A -85,B 0,C 180,E1 -11591.428,E2 -11591.428} C_VEL
LIN {X 0,Y 393.757,Z 233.975,A -85,B 0,C 180,E1 -11592.113,E2 -11592.113} C_VEL
LIN {X 0,Y 394.52,Z 244.486,A -85,B 0,C 180,E1 -11592.73,E2 -11592.73} C_VEL
LIN {X 0,Y 393.758,Z 256.362,A -85,B 0,C 180,E1 -11593.539,E2 -11593.539} C_VEL
LIN {X 0,Y 392.742,Z 268.127,A -85,B 0,C 180,E1 -11594.561,E2 -11594.561} C_VEL
LIN {X 0,Y 391.743,Z 278.005,A -85,B 0,C 180,E1 -11595.646,E2 -11595.646} C_VEL
LIN {X 0,Y 391.012,Z 286.245,A -85,B 0,C 180,E1 -11596.75,E2 -11596.75} C_VEL
LIN {X 0,Y 390.344,Z 294.302,A -85,B 0,C 180,E1 -11598.049,E2 -11598.049} C_VEL
LIN {X 0,Y 389.641,Z 302.195,A -85,B 0,C 180,E1 -11599.607,E2 -11599.607} C_VEL
LIN {X 0,Y 389.164,Z 308.476,A -85,B 0,C 180,E1 -11601.168,E2 -11601.168} C_VEL
LIN {X 0,Y 388.929,Z 313.465,A -85,B 0,C 180,E1 -11602.732,E2 -11602.732} C_VEL
LIN {X 0,Y 388.777,Z 316.348,A -85,B 0,C 180,E1 -11603.853,E2 -11603.853} C_VEL
LIN {X 0,Y 388.761,Z 318.328,A -85,B 0,C 180,E1 -11604.812,E2 -11604.812} C_VEL
LIN {X 0,Y 388.729,Z 320.047,A -85,B 0,C 180,E1 -11605.851,E2 -11605.851} C_VEL
LIN {X 0,Y 388.718,Z 321.351,A -85,B 0,C 180,E1 -11606.889,E2 -11606.889} C_VEL
LIN {X 0,Y 388.828,Z 322.19,A -85,B 0,C 180,E1 -11607.927,E2 -11607.927} C_VEL
LIN {X 0,Y 388.784,Z 322.6,A -85,B 0,C 180,E1 -11608.963,E2 -11608.963} C_VEL
LIN {X 0,Y 388.804,Z 322.607,A -85,B 0,C 180,E1 -11609.998,E2 -11609.998} C_VEL
LIN {X 0,Y 388.813,Z 322.155,A -85,B 0,C 180,E1 -11611.034,E2 -11611.034} C_VEL
LIN {X 0,Y 388.852,Z 321.269,A -85,B 0,C 180,E1 -11612.07,E2 -11612.07} C_VEL
LIN {X 0,Y 388.81,Z 319.959,A -85,B 0,C 180,E1 -11613.107,E2 -11613.107} C_VEL
LIN {X 0,Y 388.82,Z 317.1,A -85,B 0,C 180,E1 -11614.664,E2 -11614.664} C_VEL
LIN {X 0,Y 388.872,Z 312.948,A -85,B 0,C 180,E1 -11616.276,E2 -11616.276} C_VEL
LIN {X 0,Y 389.037,Z 306.841,A -85,B 0,C 180,E1 -11618.046,E2 -11618.046} C_VEL
LIN {X 0,Y 389.288,Z 299.913,A -85,B 0,C 180,E1 -11619.611,E2 -11619.611} C_VEL
LIN {X 0,Y 389.737,Z 291.113,A -85,B 0,C 180,E1 -11621.176,E2 -11621.176} C_VEL
LIN {X 0,Y 390.177,Z 282.015,A -85,B 0,C 180,E1 -11622.481,E2 -11622.481} C_VEL
LIN {X 0,Y 390.718,Z 273.109,A -85,B 0,C 180,E1 -11623.521,E2 -11623.521} C_VEL
LIN {X 0,Y 391.355,Z 262.079,A -85,B 0,C 180,E1 -11624.559,E2 -11624.559} C_VEL
LIN {X 0,Y 391.898,Z 251.672,A -85,B 0,C 180,E1 -11625.336,E2 -11625.336} C_VEL
LIN {X 0,Y 392.142,Z 241.654,A -85,B 0,C 180,E1 -11625.926,E2 -11625.926} C_VEL
LIN {X 0,Y 390.85,Z 228.704,A -85,B 0,C 180,E1 -11626.517,E2 -11626.517} C_VEL
LIN {X 0,Y 390.043,Z 220.318,A -85,B 0,C 180,E1 -11626.791,E2 -11626.791} C_VEL
LIN {X 0,Y 390.968,Z 207.647,A -85,B 0,C 180,E1 -11630.411,E2 -11630.411} C_VEL
LIN {X 0,Y 392.184,Z 194.115,A -85,B 0,C 180,E1 -11634.339,E2 -11634.339} C_VEL
LIN {X 0,Y 393.354,Z 182.826,A -85,B 0,C 180,E1 -11637.678,E2 -11637.678} C_VEL
LIN {X 0,Y 393.041,Z 178.976,A -85,B 0,C 180,E1 -11638.865,E2 -11638.865} C_VEL
LIN {X 0,Y 390.907,Z 168.38,A -85,B 0,C 180,E1 -11642.328,E2 -11642.328} C_VEL
LIN {X 0,Y 390.09,Z 163.897,A -85,B 0,C 180,E1 -11643.872,E2 -11643.872} C_VEL
LIN {X 0,Y 390.037,Z 163.899,A -85,B 0,C 180,E1 -11647.549,E2 -11647.549} C_VEL
LIN {X 0,Y 390.046,Z 163.901,A -85,B 0,C 180,E1 -11650.819,E2 -11650.819} C_VEL
LIN {X 0,Y 390.049,Z 163.897,A -85,B 0,C 180,E1 -11653.885,E2 -11653.885} C_VEL
LIN {X 0,Y 390.108,Z 163.893,A -85,B 0,C 180,E1 -11656.796,E2 -11656.796} C_VEL
LIN {X 0,Y 390.068,Z 163.896,A -85,B 0,C 180,E1 -11659.562,E2 -11659.562} C_VEL
LIN {X 0,Y 390.034,Z 163.903,A -85,B 0,C 180,E1 -11662.447,E2 -11662.447} C_VEL
LIN {X 0,Y 390.056,Z 163.901,A -85,B 0,C 180,E1 -11666.044,E2 -11666.044} C_VEL
LIN {X 0,Y 390.04,Z 163.902,A -85,B 0,C 180,E1 -11669.866,E2 -11669.866} C_VEL
LIN {X 0,Y 390.101,Z 163.892,A -85,B 0,C 180,E1 -11673.231,E2 -11673.231} C_VEL
LIN {X 0,Y 390.063,Z 163.894,A -85,B 0,C 180,E1 -11676.76,E2 -11676.76} C_VEL
LIN {X 0,Y 390.09,Z 163.894,A -85,B 0,C 180,E1 -11679.982,E2 -11679.982} C_VEL
LIN {X 0,Y 390.124,Z 163.891,A -85,B 0,C 180,E1 -11683.247,E2 -11683.247} C_VEL
LIN {X 0,Y 390.18,Z 163.881,A -85,B 0,C 180,E1 -11686.561,E2 -11686.561} C_VEL
LIN {X 0,Y 390.157,Z 163.886,A -85,B 0,C 180,E1 -11689.622,E2 -11689.622} C_VEL
LIN {X 0,Y 390.293,Z 163.868,A -85,B 0,C 180,E1 -11692.759,E2 -11692.759} C_VEL
LIN {X 0,Y 390.216,Z 163.88,A -85,B 0,C 180,E1 -11694.833,E2 -11694.833} C_VEL
LIN {X 0,Y 390.406,Z 163.853,A -85,B 0,C 180,E1 -11697.937,E2 -11697.937} C_VEL
LIN {X 0,Y 390.534,Z 163.837,A -85,B 0,C 180,E1 -11700,E2 -11700} C_VEL
LIN {X 0,Y 390.291,Z 163.87,A -85,B 0,C 180,E1 -11703.097,E2 -11703.097} C_VEL
LIN {X 0,Y 390.294,Z 163.866,A -85,B 0,C 180,E1 -11706.664,E2 -11706.664} C_VEL
LIN {X 0,Y 390.196,Z 163.88,A -85,B 0,C 180,E1 -11709.329,E2 -11709.329} C_VEL
LIN {X 0,Y 390.164,Z 163.886,A -85,B 0,C 180,E1 -11712.483,E2 -11712.483} C_VEL
LIN {X 0,Y 390.125,Z 163.887,A -85,B 0,C 180,E1 -11715.677,E2 -11715.677} C_VEL
LIN {X 0,Y 390.103,Z 163.892,A -85,B 0,C 180,E1 -11718.922,E2 -11718.922} C_VEL
LIN {X 0,Y 390.049,Z 163.9,A -85,B 0,C 180,E1 -11722.234,E2 -11722.234} C_VEL
LIN {X 0,Y 390.07,Z 163.896,A -85,B 0,C 180,E1 -11725.734,E2 -11725.734} C_VEL
LIN {X 0,Y 390.02,Z 163.9,A -85,B 0,C 180,E1 -11729.113,E2 -11729.113} C_VEL
LIN {X 0,Y 390.03,Z 163.9,A -85,B 0,C 180,E1 -11732.723,E2 -11732.723} C_VEL
LIN {X 0,Y 390.046,Z 163.901,A -85,B 0,C 180,E1 -11735.827,E2 -11735.827} C_VEL
LIN {X 0,Y 390.061,Z 163.897,A -85,B 0,C 180,E1 -11739.22,E2 -11739.22} C_VEL
LIN {X 0,Y 390.034,Z 163.899,A -85,B 0,C 180,E1 -11742.376,E2 -11742.376} C_VEL
LIN {X 0,Y 390.038,Z 163.902,A -85,B 0,C 180,E1 -11745.357,E2 -11745.357} C_VEL
LIN {X 0,Y 390.023,Z 163.901,A -85,B 0,C 180,E1 -11748.189,E2 -11748.189} C_VEL
LIN {X 0,Y 390.079,Z 163.895,A -85,B 0,C 180,E1 -11750.909,E2 -11750.909} C_VEL
LIN {X 0,Y 390.077,Z 163.896,A -85,B 0,C 180,E1 -11754.795,E2 -11754.795} C_VEL
LIN {X 0,Y 390.023,Z 163.902,A -85,B 0,C 180,E1 -11758.498,E2 -11758.498} C_VEL
LIN {X 0,Y 390.112,Z 163.89,A -85,B 0,C 180,E1 -11762.072,E2 -11762.072} C_VEL
LIN {X 0,Y 390.072,Z 163.894,A -85,B 0,C 180,E1 -11765.521,E2 -11765.521} C_VEL
LIN {X 0,Y 390.059,Z 163.899,A -85,B 0,C 180,E1 -11768.88,E2 -11768.88} C_VEL
LIN {X 0,Y 390.126,Z 163.89,A -85,B 0,C 180,E1 -11772.169,E2 -11772.169} C_VEL
LIN {X 0,Y 390.141,Z 163.886,A -85,B 0,C 180,E1 -11775.394,E2 -11775.394} C_VEL
LIN {X 0,Y 390.146,Z 163.888,A -85,B 0,C 180,E1 -11778.573,E2 -11778.573} C_VEL
LIN {X 0,Y 390.344,Z 163.864,A -85,B 0,C 180,E1 -11781.995,E2 -11781.995} C_VEL
LIN {X 0,Y 390.228,Z 163.876,A -85,B 0,C 180,E1 -11784.835,E2 -11784.835} C_VEL
LIN {X 0,Y 390.419,Z 163.854,A -85,B 0,C 180,E1 -11787.938,E2 -11787.938} C_VEL
LIN {X 0,Y 390.417,Z 163.854,A -85,B 0,C 180,E1 -11792.065,E2 -11792.065} C_VEL
LIN {X 0,Y 390.333,Z 163.865,A -85,B 0,C 180,E1 -11796.203,E2 -11796.203} C_VEL
LIN {X 0,Y 390.318,Z 163.865,A -85,B 0,C 180,E1 -11798.284,E2 -11798.284} C_VEL
LIN {X 0,Y 390.174,Z 163.881,A -85,B 0,C 180,E1 -11802.484,E2 -11802.484} C_VEL
LIN {X 0,Y 390.141,Z 163.888,A -85,B 0,C 180,E1 -11805.678,E2 -11805.678} C_VEL
LIN {X 0,Y 390.109,Z 163.892,A -85,B 0,C 180,E1 -11808.923,E2 -11808.923} C_VEL
LIN {X 0,Y 390.039,Z 163.899,A -85,B 0,C 180,E1 -11812.236,E2 -11812.236} C_VEL
LIN {X 0,Y 390.054,Z 163.896,A -85,B 0,C 180,E1 -11815.723,E2 -11815.723} C_VEL
LIN {X 0,Y 390.03,Z 163.903,A -85,B 0,C 180,E1 -11819.113,E2 -11819.113} C_VEL
LIN {X 0,Y 390.014,Z 163.9,A -85,B 0,C 180,E1 -11820.829,E2 -11820.829} C_VEL
LIN {X 0,Y 389.343,Z 163.987,A -85,B 0,C 180,E1 -11821.691,E2 -11821.691} C_VEL
LIN {X 0,Y 386.496,Z 164.343,A -85,B 0,C 180,E1 -11823.093,E2 -11823.093} C_VEL
LIN {X 0,Y 384.097,Z 164.64,A -85,B 0,C 180,E1 -11824.226,E2 -11824.226} C_VEL
LIN {X 0,Y 383.079,Z 164.769,A -85,B 0,C 180,E1 -11825.101,E2 -11825.101} C_VEL
LIN {X 0,Y 383.002,Z 164.773,A -85,B 0,C 180,E1 -11825.398,E2 -11825.398} C_VEL
LIN {X 0,Y 382.985,Z 164.781,A -85,B 0,C 180,E1 -11828.604,E2 -11828.604} C_VEL
LIN {X 0,Y 382.966,Z 164.78,A -85,B 0,C 180,E1 -11831.351,E2 -11831.351} C_VEL
LIN {X 0,Y 383,Z 164.779,A -85,B 0,C 180,E1 -11834.304,E2 -11834.304} C_VEL
LIN {X 0,Y 383.016,Z 164.774,A -85,B 0,C 180,E1 -11837.241,E2 -11837.241} C_VEL
LIN {X 0,Y 383.003,Z 164.779,A -85,B 0,C 180,E1 -11840.417,E2 -11840.417} C_VEL
LIN {X 0,Y 383.028,Z 164.776,A -85,B 0,C 180,E1 -11844.045,E2 -11844.045} C_VEL
LIN {X 0,Y 383.11,Z 164.925,A -85,B 0,C 180,E1 -11846.532,E2 -11846.532} C_VEL
LIN {X 0,Y 384.008,Z 170.793,A -85,B 0,C 180,E1 -11849.339,E2 -11849.339} C_VEL
LIN {X 0,Y 383.769,Z 176.97,A -85,B 0,C 180,E1 -11852.161,E2 -11852.161} C_VEL
LIN {X 0,Y 383.291,Z 184.74,A -85,B 0,C 180,E1 -11855.634,E2 -11855.634} C_VEL
LIN {X 0,Y 382.834,Z 193.739,A -85,B 0,C 180,E1 -11859.586,E2 -11859.586} C_VEL
LIN {X 0,Y 382.494,Z 201.392,A -85,B 0,C 180,E1 -11862.903,E2 -11862.903} C_VEL
LIN {X 0,Y 382.219,Z 209.034,A -85,B 0,C 180,E1 -11866.17,E2 -11866.17} C_VEL
LIN {X 0,Y 382.059,Z 215.715,A -85,B 0,C 180,E1 -11868.998,E2 -11868.998} C_VEL
LIN {X 0,Y 383.047,Z 226.673,A -85,B 0,C 180,E1 -11869.628,E2 -11869.628} C_VEL
LIN {X 0,Y 383.618,Z 234.841,A -85,B 0,C 180,E1 -11870.243,E2 -11870.243} C_VEL
LIN {X 0,Y 383.154,Z 244.609,A -85,B 0,C 180,E1 -11871.163,E2 -11871.163} C_VEL
LIN {X 0,Y 382.836,Z 252.289,A -85,B 0,C 180,E1 -11872.086,E2 -11872.086} C_VEL
LIN {X 0,Y 382.489,Z 259.393,A -85,B 0,C 180,E1 -11873.145,E2 -11873.145} C_VEL
LIN {X 0,Y 382.296,Z 266.328,A -85,B 0,C 180,E1 -11874.462,E2 -11874.462} C_VEL
LIN {X 0,Y 382.042,Z 271.658,A -85,B 0,C 180,E1 -11875.78,E2 -11875.78} C_VEL
LIN {X 0,Y 381.874,Z 276.27,A -85,B 0,C 180,E1 -11877.363,E2 -11877.363} C_VEL
LIN {X 0,Y 381.75,Z 279.207,A -85,B 0,C 180,E1 -11878.945,E2 -11878.945} C_VEL
LIN {X 0,Y 381.743,Z 280.309,A -85,B 0,C 180,E1 -11880,E2 -11880} C_VEL
LIN {X 0,Y 381.824,Z 280.745,A -85,B 0,C 180,E1 -11881.055,E2 -11881.055} C_VEL
LIN {X 0,Y 381.98,Z 280.517,A -85,B 0,C 180,E1 -11882.109,E2 -11882.109} C_VEL
LIN {X 0,Y 382.227,Z 279.627,A -85,B 0,C 180,E1 -11883.162,E2 -11883.162} C_VEL
LIN {X 0,Y 382.627,Z 278.059,A -85,B 0,C 180,E1 -11884.213,E2 -11884.213} C_VEL
LIN {X 0,Y 382.853,Z 274.439,A -85,B 0,C 180,E1 -11885.795,E2 -11885.795} C_VEL
LIN {X 0,Y 383.393,Z 269.083,A -85,B 0,C 180,E1 -11887.372,E2 -11887.372} C_VEL
LIN {X 0,Y 384.155,Z 263.057,A -85,B 0,C 180,E1 -11888.681,E2 -11888.681} C_VEL
LIN {X 0,Y 385.119,Z 255.616,A -85,B 0,C 180,E1 -11889.931,E2 -11889.931} C_VEL
LIN {X 0,Y 386.008,Z 247.401,A -85,B 0,C 180,E1 -11891.021,E2 -11891.021} C_VEL
LIN {X 0,Y 386.764,Z 238.855,A -85,B 0,C 180,E1 -11891.929,E2 -11891.929} C_VEL
LIN {X 0,Y 385.556,Z 228.772,A -85,B 0,C 180,E1 -11892.91,E2 -11892.91} C_VEL
LIN {X 0,Y 382.989,Z 217.055,A -85,B 0,C 180,E1 -11893.903,E2 -11893.903} C_VEL
LIN {X 0,Y 383.609,Z 209.065,A -85,B 0,C 180,E1 -11897.694,E2 -11897.694} C_VEL
LIN {X 0,Y 384.289,Z 201.519,A -85,B 0,C 180,E1 -11901.455,E2 -11901.455} C_VEL
LIN {X 0,Y 385.201,Z 194.134,A -85,B 0,C 180,E1 -11905.389,E2 -11905.389} C_VEL
LIN {X 0,Y 386.331,Z 187.613,A -85,B 0,C 180,E1 -11909.165,E2 -11909.165} C_VEL
LIN {X 0,Y 386.741,Z 184.325,A -85,B 0,C 180,E1 -11911.338,E2 -11911.338} C_VEL
LIN {X 0,Y 386.617,Z 181.846,A -85,B 0,C 180,E1 -11913.257,E2 -11913.257} C_VEL
LIN {X 0,Y 386.214,Z 179.296,A -85,B 0,C 180,E1 -11915.613,E2 -11915.613} C_VEL
LIN {X 0,Y 385.851,Z 176.913,A -85,B 0,C 180,E1 -11918.442,E2 -11918.442} C_VEL
LIN {X 0,Y 385.586,Z 175.498,A -85,B 0,C 180,E1 -11921.008,E2 -11921.008} C_VEL
LIN {X 0,Y 385.474,Z 174.781,A -85,B 0,C 180,E1 -11923.854,E2 -11923.854} C_VEL
LIN {X 0,Y 385.597,Z 175.086,A -85,B 0,C 180,E1 -11926.807,E2 -11926.807} C_VEL
LIN {X 0,Y 385.971,Z 176.628,A -85,B 0,C 180,E1 -11929.886,E2 -11929.886} C_VEL
LIN {X 0,Y 386.359,Z 178.199,A -85,B 0,C 180,E1 -11931.794,E2 -11931.794} C_VEL
LIN {X 0,Y 387.112,Z 181.621,A -85,B 0,C 180,E1 -11934.783,E2 -11934.783} C_VEL
LIN {X 0,Y 388.076,Z 186.066,A -85,B 0,C 180,E1 -11937.707,E2 -11937.707} C_VEL
LIN {X 0,Y 388.863,Z 190.681,A -85,B 0,C 180,E1 -11940.172,E2 -11940.172} C_VEL
LIN {X 0,Y 388.958,Z 193.317,A -85,B 0,C 180,E1 -11941.39,E2 -11941.39} C_VEL
LIN {X 0,Y 387.416,Z 200.552,A -85,B 0,C 180,E1 -11944.189,E2 -11944.189} C_VEL
LIN {X 0,Y 385.447,Z 211.697,A -85,B 0,C 180,E1 -11948.106,E2 -11948.106} C_VEL
LIN {X 0,Y 384.367,Z 220.606,A -85,B 0,C 180,E1 -11950.956,E2 -11950.956} C_VEL
LIN {X 0,Y 386.941,Z 233.336,A -85,B 0,C 180,E1 -11951.642,E2 -11951.642} C_VEL
LIN {X 0,Y 387.774,Z 242.7,A -85,B 0,C 180,E1 -11952.21,E2 -11952.21} C_VEL
LIN {X 0,Y 387.629,Z 250.591,A -85,B 0,C 180,E1 -11952.736,E2 -11952.736} C_VEL
LIN {X 0,Y 386.634,Z 261.988,A -85,B 0,C 180,E1 -11953.634,E2 -11953.634} C_VEL
LIN {X 0,Y 385.558,Z 272.465,A -85,B 0,C 180,E1 -11954.673,E2 -11954.673} C_VEL
LIN {X 0,Y 384.487,Z 281.798,A -85,B 0,C 180,E1 -11955.821,E2 -11955.821} C_VEL
LIN {X 0,Y 383.746,Z 291.501,A -85,B 0,C 180,E1 -11957.303,E2 -11957.303} C_VEL
LIN {X 0,Y 382.781,Z 299.81,A -85,B 0,C 180,E1 -11958.883,E2 -11958.883} C_VEL
LIN {X 0,Y 382.288,Z 306.502,A -85,B 0,C 180,E1 -11960.475,E2 -11960.475} C_VEL
LIN {X 0,Y 381.911,Z 311.838,A -85,B 0,C 180,E1 -11962.065,E2 -11962.065} C_VEL
LIN {X 0,Y 381.683,Z 316.446,A -85,B 0,C 180,E1 -11963.888,E2 -11963.888} C_VEL
LIN {X 0,Y 381.653,Z 319.767,A -85,B 0,C 180,E1 -11965.774,E2 -11965.774} C_VEL
LIN {X 0,Y 381.623,Z 321.022,A -85,B 0,C 180,E1 -11966.831,E2 -11966.831} C_VEL
LIN {X 0,Y 381.74,Z 321.815,A -85,B 0,C 180,E1 -11967.888,E2 -11967.888} C_VEL
LIN {X 0,Y 381.715,Z 322.195,A -85,B 0,C 180,E1 -11968.943,E2 -11968.943} C_VEL
LIN {X 0,Y 381.73,Z 322.161,A -85,B 0,C 180,E1 -11969.998,E2 -11969.998} C_VEL
LIN {X 0,Y 381.742,Z 321.655,A -85,B 0,C 180,E1 -11971.053,E2 -11971.053} C_VEL
LIN {X 0,Y 381.785,Z 320.736,A -85,B 0,C 180,E1 -11972.108,E2 -11972.108} C_VEL
LIN {X 0,Y 381.717,Z 319.375,A -85,B 0,C 180,E1 -11973.165,E2 -11973.165} C_VEL
LIN {X 0,Y 381.755,Z 316.428,A -85,B 0,C 180,E1 -11974.75,E2 -11974.75} C_VEL
LIN {X 0,Y 381.807,Z 312.333,A -85,B 0,C 180,E1 -11976.339,E2 -11976.339} C_VEL
LIN {X 0,Y 381.989,Z 305.966,A -85,B 0,C 180,E1 -11978.196,E2 -11978.196} C_VEL
LIN {X 0,Y 382.224,Z 298.861,A -85,B 0,C 180,E1 -11979.791,E2 -11979.791} C_VEL
LIN {X 0,Y 382.723,Z 289.924,A -85,B 0,C 180,E1 -11981.383,E2 -11981.383} C_VEL
LIN {X 0,Y 383.229,Z 280.585,A -85,B 0,C 180,E1 -11982.711,E2 -11982.711} C_VEL
LIN {X 0,Y 383.708,Z 271.418,A -85,B 0,C 180,E1 -11983.773,E2 -11983.773} C_VEL
LIN {X 0,Y 384.499,Z 260.139,A -85,B 0,C 180,E1 -11984.825,E2 -11984.825} C_VEL
LIN {X 0,Y 384.982,Z 249.234,A -85,B 0,C 180,E1 -11985.619,E2 -11985.619} C_VEL
LIN {X 0,Y 385.056,Z 241.138,A -85,B 0,C 180,E1 -11986.091,E2 -11986.091} C_VEL
LIN {X 0,Y 383.713,Z 228.418,A -85,B 0,C 180,E1 -11986.679,E2 -11986.679} C_VEL
LIN {X 0,Y 383.007,Z 220.263,A -85,B 0,C 180,E1 -11986.968,E2 -11986.968} C_VEL
LIN {X 0,Y 383.953,Z 207.483,A -85,B 0,C 180,E1 -11990.696,E2 -11990.696} C_VEL
LIN {X 0,Y 385.156,Z 194.959,A -85,B 0,C 180,E1 -11994.41,E2 -11994.41} C_VEL
LIN {X 0,Y 386.317,Z 184.238,A -85,B 0,C 180,E1 -11997.637,E2 -11997.637} C_VEL
LIN {X 0,Y 385.963,Z 179.732,A -85,B 0,C 180,E1 -11999.069,E2 -11999.069} C_VEL
LIN {X 0,Y 383.824,Z 169.084,A -85,B 0,C 180,E1 -12002.618,E2 -12002.618} C_VEL
LIN {X 0,Y 383.028,Z 164.776,A -85,B 0,C 180,E1 -12004.131,E2 -12004.131} C_VEL
LIN {X 0,Y 382.989,Z 164.778,A -85,B 0,C 180,E1 -12007.267,E2 -12007.267} C_VEL
LIN {X 0,Y 382.999,Z 164.775,A -85,B 0,C 180,E1 -12009.957,E2 -12009.957} C_VEL
LIN {X 0,Y 382.997,Z 164.778,A -85,B 0,C 180,E1 -12012.777,E2 -12012.777} C_VEL
LIN {X 0,Y 383.032,Z 164.772,A -85,B 0,C 180,E1 -12015.794,E2 -12015.794} C_VEL
LIN {X 0,Y 383.035,Z 164.773,A -85,B 0,C 180,E1 -12018.785,E2 -12018.785} C_VEL
LIN {X 0,Y 382.991,Z 164.779,A -85,B 0,C 180,E1 -12022.094,E2 -12022.094} C_VEL
LIN {X 0,Y 383.006,Z 164.774,A -85,B 0,C 180,E1 -12025.331,E2 -12025.331} C_VEL
LIN {X 0,Y 382.974,Z 164.779,A -85,B 0,C 180,E1 -12029.08,E2 -12029.08} C_VEL
LIN {X 0,Y 383.044,Z 164.77,A -85,B 0,C 180,E1 -12032.697,E2 -12032.697} C_VEL
LIN {X 0,Y 383.037,Z 164.77,A -85,B 0,C 180,E1 -12035.039,E2 -12035.039} C_VEL
LIN {X 0,Y 382.978,Z 164.778,A -85,B 0,C 180,E1 -12038.468,E2 -12038.468} C_VEL
LIN {X 0,Y 383.075,Z 164.769,A -85,B 0,C 180,E1 -12041.827,E2 -12041.827} C_VEL
LIN {X 0,Y 383.098,Z 164.766,A -85,B 0,C 180,E1 -12045.118,E2 -12045.118} C_VEL
LIN {X 0,Y 383.09,Z 164.763,A -85,B 0,C 180,E1 -12048.358,E2 -12048.358} C_VEL
LIN {X 0,Y 383.25,Z 164.744,A -85,B 0,C 180,E1 -12051.974,E2 -12051.974} C_VEL
LIN {X 0,Y 383.188,Z 164.754,A -85,B 0,C 180,E1 -12054.738,E2 -12054.738} C_VEL
LIN {X 0,Y 383.374,Z 164.729,A -85,B 0,C 180,E1 -12057.899,E2 -12057.899} C_VEL
LIN {X 0,Y 383.504,Z 164.712,A -85,B 0,C 180,E1 -12060,E2 -12060} C_VEL
LIN {X 0,Y 383.228,Z 164.749,A -85,B 0,C 180,E1 -12063.154,E2 -12063.154} C_VEL
LIN {X 0,Y 383.253,Z 164.744,A -85,B 0,C 180,E1 -12066.659,E2 -12066.659} C_VEL
LIN {X 0,Y 383.246,Z 164.748,A -85,B 0,C 180,E1 -12068.436,E2 -12068.436} C_VEL
LIN {X 0,Y 383.093,Z 164.764,A -85,B 0,C 180,E1 -12071.642,E2 -12071.642} C_VEL
LIN {X 0,Y 383.098,Z 164.764,A -85,B 0,C 180,E1 -12074.882,E2 -12074.882} C_VEL
LIN {X 0,Y 383.08,Z 164.769,A -85,B 0,C 180,E1 -12078.173,E2 -12078.173} C_VEL
LIN {X 0,Y 383,Z 164.776,A -85,B 0,C 180,E1 -12081.531,E2 -12081.531} C_VEL
LIN {X 0,Y 383.018,Z 164.773,A -85,B 0,C 180,E1 -12084.963,E2 -12084.963} C_VEL
LIN {X 0,Y 382.973,Z 164.78,A -85,B 0,C 180,E1 -12088.498,E2 -12088.498} C_VEL
LIN {X 0,Y 382.997,Z 164.778,A -85,B 0,C 180,E1 -12092.151,E2 -12092.151} C_VEL
LIN {X 0,Y 383.006,Z 164.775,A -85,B 0,C 180,E1 -12094.669,E2 -12094.669} C_VEL
LIN {X 0,Y 382.991,Z 164.78,A -85,B 0,C 180,E1 -12097.906,E2 -12097.906} C_VEL
LIN {X 0,Y 382.974,Z 164.781,A -85,B 0,C 180,E1 -12101.349,E2 -12101.349} C_VEL
LIN {X 0,Y 382.989,Z 164.777,A -85,B 0,C 180,E1 -12104.305,E2 -12104.305} C_VEL
LIN {X 0,Y 383.001,Z 164.778,A -85,B 0,C 180,E1 -12107.242,E2 -12107.242} C_VEL
LIN {X 0,Y 383.005,Z 164.774,A -85,B 0,C 180,E1 -12110.415,E2 -12110.415} C_VEL
LIN {X 0,Y 383.017,Z 164.772,A -85,B 0,C 180,E1 -12114.046,E2 -12114.046} C_VEL
LIN {X 0,Y 382.982,Z 164.779,A -85,B 0,C 180,E1 -12117.579,E2 -12117.579} C_VEL
LIN {X 0,Y 382.993,Z 164.777,A -85,B 0,C 180,E1 -12120.303,E2 -12120.303} C_VEL
LIN {X 0,Y 383.051,Z 164.771,A -85,B 0,C 180,E1 -12122.7,E2 -12122.7} C_VEL
LIN {X 0,Y 383.028,Z 164.772,A -85,B 0,C 180,E1 -12126.194,E2 -12126.194} C_VEL
LIN {X 0,Y 383.053,Z 164.769,A -85,B 0,C 180,E1 -12129.6,E2 -12129.6} C_VEL
LIN {X 0,Y 383.103,Z 164.765,A -85,B 0,C 180,E1 -12132.933,E2 -12132.933} C_VEL
LIN {X 0,Y 383.124,Z 164.764,A -85,B 0,C 180,E1 -12136.466,E2 -12136.466} C_VEL
LIN {X 0,Y 383.15,Z 164.759,A -85,B 0,C 180,E1 -12140.5,E2 -12140.5} C_VEL
LIN {X 0,Y 383.274,Z 164.744,A -85,B 0,C 180,E1 -12142.627,E2 -12142.627} C_VEL
LIN {X 0,Y 383.2,Z 164.752,A -85,B 0,C 180,E1 -12144.74,E2 -12144.74} C_VEL
LIN {X 0,Y 383.387,Z 164.73,A -85,B 0,C 180,E1 -12147.901,E2 -12147.901} C_VEL
LIN {X 0,Y 383.384,Z 164.73,A -85,B 0,C 180,E1 -12152.103,E2 -12152.103} C_VEL
LIN {X 0,Y 383.29,Z 164.741,A -85,B 0,C 180,E1 -12156.318,E2 -12156.318} C_VEL
LIN {X 0,Y 383.263,Z 164.743,A -85,B 0,C 180,E1 -12158.437,E2 -12158.437} C_VEL
LIN {X 0,Y 383.101,Z 164.767,A -85,B 0,C 180,E1 -12161.644,E2 -12161.644} C_VEL
LIN {X 0,Y 383.112,Z 164.761,A -85,B 0,C 180,E1 -12164.883,E2 -12164.883} C_VEL
LIN {X 0,Y 383.067,Z 164.767,A -85,B 0,C 180,E1 -12168.175,E2 -12168.175} C_VEL
LIN {X 0,Y 382.995,Z 164.78,A -85,B 0,C 180,E1 -12171.532,E2 -12171.532} C_VEL
LIN {X 0,Y 382.99,Z 164.779,A -85,B 0,C 180,E1 -12174.966,E2 -12174.966} C_VEL
LIN {X 0,Y 382.98,Z 164.779,A -85,B 0,C 180,E1 -12178.499,E2 -12178.499} C_VEL
LIN {X 0,Y 383.014,Z 164.774,A -85,B 0,C 180,E1 -12182.151,E2 -12182.151} C_VEL
LIN {X 0,Y 383.002,Z 164.773,A -85,B 0,C 180,E1 -12185.398,E2 -12185.398} C_VEL
LIN {X 0,Y 382.356,Z 164.857,A -85,B 0,C 180,E1 -12186.276,E2 -12186.276} C_VEL
LIN {X 0,Y 379.526,Z 165.208,A -85,B 0,C 180,E1 -12187.703,E2 -12187.703} C_VEL
LIN {X 0,Y 377.102,Z 165.513,A -85,B 0,C 180,E1 -12188.856,E2 -12188.856} C_VEL
LIN {X 0,Y 376.036,Z 165.643,A -85,B 0,C 180,E1 -12189.748,E2 -12189.748} C_VEL
LIN {X 0,Y 375.936,Z 165.654,A -85,B 0,C 180,E1 -12190.05,E2 -12190.05} C_VEL
LIN {X 0,Y 375.934,Z 165.656,A -85,B 0,C 180,E1 -12193.767,E2 -12193.767} C_VEL
LIN {X 0,Y 375.94,Z 165.657,A -85,B 0,C 180,E1 -12196.811,E2 -12196.811} C_VEL
LIN {X 0,Y 375.95,Z 165.656,A -85,B 0,C 180,E1 -12200.536,E2 -12200.536} C_VEL
LIN {X 0,Y 375.967,Z 165.651,A -85,B 0,C 180,E1 -12203.497,E2 -12203.497} C_VEL
LIN {X 0,Y 376.067,Z 165.748,A -85,B 0,C 180,E1 -12206.384,E2 -12206.384} C_VEL
LIN {X 0,Y 376.947,Z 171.236,A -85,B 0,C 180,E1 -12209.056,E2 -12209.056} C_VEL
LIN {X 0,Y 376.824,Z 175.917,A -85,B 0,C 180,E1 -12211.234,E2 -12211.234} C_VEL
LIN {X 0,Y 376.379,Z 183.221,A -85,B 0,C 180,E1 -12214.566,E2 -12214.566} C_VEL
LIN {X 0,Y 375.877,Z 192.25,A -85,B 0,C 180,E1 -12218.617,E2 -12218.617} C_VEL
LIN {X 0,Y 375.487,Z 201.224,A -85,B 0,C 180,E1 -12222.574,E2 -12222.574} C_VEL
LIN {X 0,Y 375.128,Z 210.179,A -85,B 0,C 180,E1 -12226.457,E2 -12226.457} C_VEL
LIN {X 0,Y 374.961,Z 215.771,A -85,B 0,C 180,E1 -12228.855,E2 -12228.855} C_VEL
LIN {X 0,Y 375.914,Z 226.59,A -85,B 0,C 180,E1 -12229.497,E2 -12229.497} C_VEL
LIN {X 0,Y 376.58,Z 233.997,A -85,B 0,C 180,E1 -12230.059,E2 -12230.059} C_VEL
LIN {X 0,Y 376.101,Z 243.998,A -85,B 0,C 180,E1 -12230.996,E2 -12230.996} C_VEL
LIN {X 0,Y 375.79,Z 251.87,A -85,B 0,C 180,E1 -12231.937,E2 -12231.937} C_VEL
LIN {X 0,Y 375.395,Z 259.965,A -85,B 0,C 180,E1 -12233.161,E2 -12233.161} C_VEL
LIN {X 0,Y 375.223,Z 266.196,A -85,B 0,C 180,E1 -12234.357,E2 -12234.357} C_VEL
LIN {X 0,Y 374.961,Z 271.65,A -85,B 0,C 180,E1 -12235.7,E2 -12235.7} C_VEL
LIN {X 0,Y 374.793,Z 276.402,A -85,B 0,C 180,E1 -12237.313,E2 -12237.313} C_VEL
LIN {X 0,Y 374.682,Z 279.47,A -85,B 0,C 180,E1 -12238.925,E2 -12238.925} C_VEL
LIN {X 0,Y 374.671,Z 280.658,A -85,B 0,C 180,E1 -12240,E2 -12240} C_VEL
LIN {X 0,Y 374.753,Z 281.18,A -85,B 0,C 180,E1 -12241.075,E2 -12241.075} C_VEL
LIN {X 0,Y 374.914,Z 281.034,A -85,B 0,C 180,E1 -12242.149,E2 -12242.149} C_VEL
LIN {X 0,Y 375.171,Z 280.225,A -85,B 0,C 180,E1 -12243.222,E2 -12243.222} C_VEL
LIN {X 0,Y 375.6,Z 278.749,A -85,B 0,C 180,E1 -12244.292,E2 -12244.292} C_VEL
LIN {X 0,Y 375.844,Z 275.297,A -85,B 0,C 180,E1 -12245.903,E2 -12245.903} C_VEL
LIN {X 0,Y 376.452,Z 270.147,A -85,B 0,C 180,E1 -12247.509,E2 -12247.509} C_VEL
LIN {X 0,Y 377.278,Z 264.221,A -85,B 0,C 180,E1 -12248.862,E2 -12248.862} C_VEL
LIN {X 0,Y 378.302,Z 256.824,A -85,B 0,C 180,E1 -12250.165,E2 -12250.165} C_VEL
LIN {X 0,Y 379.339,Z 248.234,A -85,B 0,C 180,E1 -12251.353,E2 -12251.353} C_VEL
LIN {X 0,Y 380.109,Z 239.871,A -85,B 0,C 180,E1 -12252.277,E2 -12252.277} C_VEL
LIN {X 0,Y 379.023,Z 230.481,A -85,B 0,C 180,E1 -12253.244,E2 -12253.244} C_VEL
LIN {X 0,Y 376.902,Z 220.493,A -85,B 0,C 180,E1 -12254.152,E2 -12254.152} C_VEL
LIN {X 0,Y 376.096,Z 217.127,A -85,B 0,C 180,E1 -12254.46,E2 -12254.46} C_VEL
LIN {X 0,Y 376.66,Z 210.081,A -85,B 0,C 180,E1 -12257.896,E2 -12257.896} C_VEL
LIN {X 0,Y 377.445,Z 202.356,A -85,B 0,C 180,E1 -12261.864,E2 -12261.864} C_VEL
LIN {X 0,Y 378.431,Z 195.096,A -85,B 0,C 180,E1 -12265.876,E2 -12265.876} C_VEL
LIN {X 0,Y 379.568,Z 189.092,A -85,B 0,C 180,E1 -12269.511,E2 -12269.511} C_VEL
LIN {X 0,Y 379.955,Z 185.957,A -85,B 0,C 180,E1 -12271.693,E2 -12271.693} C_VEL
LIN {X 0,Y 379.762,Z 183.509,A -85,B 0,C 180,E1 -12273.724,E2 -12273.724} C_VEL
LIN {X 0,Y 379.394,Z 180.936,A -85,B 0,C 180,E1 -12276.355,E2 -12276.355} C_VEL
LIN {X 0,Y 379.117,Z 178.929,A -85,B 0,C 180,E1 -12279.071,E2 -12279.071} C_VEL
LIN {X 0,Y 378.851,Z 177.644,A -85,B 0,C 180,E1 -12282.093,E2 -12282.093} C_VEL
LIN {X 0,Y 378.879,Z 177.372,A -85,B 0,C 180,E1 -12285.179,E2 -12285.179} C_VEL
LIN {X 0,Y 379.108,Z 178.198,A -85,B 0,C 180,E1 -12288.133,E2 -12288.133} C_VEL
LIN {X 0,Y 379.609,Z 180.076,A -85,B 0,C 180,E1 -12291.04,E2 -12291.04} C_VEL
LIN {X 0,Y 380.343,Z 183.615,A -85,B 0,C 180,E1 -12294.394,E2 -12294.394} C_VEL
LIN {X 0,Y 381.136,Z 187.367,A -85,B 0,C 180,E1 -12297.044,E2 -12297.044} C_VEL
LIN {X 0,Y 382.024,Z 192.285,A -85,B 0,C 180,E1 -12299.843,E2 -12299.843} C_VEL
LIN {X 0,Y 382.127,Z 195.643,A -85,B 0,C 180,E1 -12301.431,E2 -12301.431} C_VEL
LIN {X 0,Y 380.435,Z 202.787,A -85,B 0,C 180,E1 -12304.269,E2 -12304.269} C_VEL
LIN {X 0,Y 378.444,Z 213.789,A -85,B 0,C 180,E1 -12308.209,E2 -12308.209} C_VEL
LIN {X 0,Y 377.551,Z 220.387,A -85,B 0,C 180,E1 -12310.422,E2 -12310.422} C_VEL
LIN {X 0,Y 380.264,Z 233.562,A -85,B 0,C 180,E1 -12311.186,E2 -12311.186} C_VEL
LIN {X 0,Y 381.161,Z 242.018,A -85,B 0,C 180,E1 -12311.731,E2 -12311.731} C_VEL
LIN {X 0,Y 381.091,Z 250.047,A -85,B 0,C 180,E1 -12312.283,E2 -12312.283} C_VEL
LIN {X 0,Y 380.048,Z 261.521,A -85,B 0,C 180,E1 -12313.204,E2 -12313.204} C_VEL
LIN {X 0,Y 378.907,Z 271.982,A -85,B 0,C 180,E1 -12314.259,E2 -12314.259} C_VEL
LIN {X 0,Y 377.559,Z 282.799,A -85,B 0,C 180,E1 -12315.633,E2 -12315.633} C_VEL
LIN {X 0,Y 376.823,Z 291.762,A -85,B 0,C 180,E1 -12317.066,E2 -12317.066} C_VEL
LIN {X 0,Y 375.809,Z 299.921,A -85,B 0,C 180,E1 -12318.674,E2 -12318.674} C_VEL
LIN {X 0,Y 375.265,Z 306.515,A -85,B 0,C 180,E1 -12320.295,E2 -12320.295} C_VEL
LIN {X 0,Y 374.852,Z 311.735,A -85,B 0,C 180,E1 -12321.915,E2 -12321.915} C_VEL
LIN {X 0,Y 374.594,Z 316.549,A -85,B 0,C 180,E1 -12323.918,E2 -12323.918} C_VEL
LIN {X 0,Y 374.577,Z 319.498,A -85,B 0,C 180,E1 -12325.694,E2 -12325.694} C_VEL
LIN {X 0,Y 374.532,Z 320.682,A -85,B 0,C 180,E1 -12326.771,E2 -12326.771} C_VEL
LIN {X 0,Y 374.639,Z 321.441,A -85,B 0,C 180,E1 -12327.848,E2 -12327.848} C_VEL
LIN {X 0,Y 374.647,Z 321.791,A -85,B 0,C 180,E1 -12328.923,E2 -12328.923} C_VEL
LIN {X 0,Y 374.659,Z 321.687,A -85,B 0,C 180,E1 -12329.998,E2 -12329.998} C_VEL
LIN {X 0,Y 374.674,Z 321.142,A -85,B 0,C 180,E1 -12331.073,E2 -12331.073} C_VEL
LIN {X 0,Y 374.718,Z 320.188,A -85,B 0,C 180,E1 -12332.148,E2 -12332.148} C_VEL
LIN {X 0,Y 374.629,Z 318.748,A -85,B 0,C 180,E1 -12333.225,E2 -12333.225} C_VEL
LIN {X 0,Y 374.688,Z 315.718,A -85,B 0,C 180,E1 -12334.84,E2 -12334.84} C_VEL
LIN {X 0,Y 374.721,Z 311.528,A -85,B 0,C 180,E1 -12336.459,E2 -12336.459} C_VEL
LIN {X 0,Y 374.881,Z 306.069,A -85,B 0,C 180,E1 -12338.081,E2 -12338.081} C_VEL
LIN {X 0,Y 375.118,Z 299.127,A -85,B 0,C 180,E1 -12339.706,E2 -12339.706} C_VEL
LIN {X 0,Y 375.594,Z 290.315,A -85,B 0,C 180,E1 -12341.329,E2 -12341.329} C_VEL
LIN {X 0,Y 376.062,Z 281.186,A -85,B 0,C 180,E1 -12342.683,E2 -12342.683} C_VEL
LIN {X 0,Y 376.58,Z 273.242,A -85,B 0,C 180,E1 -12343.652,E2 -12343.652} C_VEL
LIN {X 0,Y 377.277,Z 261.474,A -85,B 0,C 180,E1 -12344.811,E2 -12344.811} C_VEL
LIN {X 0,Y 377.915,Z 249.736,A -85,B 0,C 180,E1 -12345.711,E2 -12345.711} C_VEL
LIN {X 0,Y 378.03,Z 241.786,A -85,B 0,C 180,E1 -12346.191,E2 -12346.191} C_VEL
LIN {X 0,Y 376.718,Z 229.07,A -85,B 0,C 180,E1 -12346.806,E2 -12346.806} C_VEL
LIN {X 0,Y 375.981,Z 220.248,A -85,B 0,C 180,E1 -12347.12,E2 -12347.12} C_VEL
LIN {X 0,Y 376.889,Z 208.117,A -85,B 0,C 180,E1 -12350.748,E2 -12350.748} C_VEL
LIN {X 0,Y 378.094,Z 196.128,A -85,B 0,C 180,E1 -12354.382,E2 -12354.382} C_VEL
LIN {X 0,Y 379.277,Z 185.666,A -85,B 0,C 180,E1 -12357.595,E2 -12357.595} C_VEL
LIN {X 0,Y 379.127,Z 181.843,A -85,B 0,C 180,E1 -12358.812,E2 -12358.812} C_VEL
LIN {X 0,Y 377.192,Z 172.215,A -85,B 0,C 180,E1 -12362.072,E2 -12362.072} C_VEL
LIN {X 0,Y 375.971,Z 165.656,A -85,B 0,C 180,E1 -12364.386,E2 -12364.386} C_VEL
LIN {X 0,Y 375.956,Z 165.653,A -85,B 0,C 180,E1 -12368.087,E2 -12368.087} C_VEL
LIN {X 0,Y 375.93,Z 165.659,A -85,B 0,C 180,E1 -12370.866,E2 -12370.866} C_VEL
LIN {X 0,Y 375.96,Z 165.655,A -85,B 0,C 180,E1 -12374.736,E2 -12374.736} C_VEL
LIN {X 0,Y 375.98,Z 165.653,A -85,B 0,C 180,E1 -12378.388,E2 -12378.388} C_VEL
LIN {X 0,Y 375.955,Z 165.655,A -85,B 0,C 180,E1 -12381.91,E2 -12381.91} C_VEL
LIN {X 0,Y 375.968,Z 165.65,A -85,B 0,C 180,E1 -12385.331,E2 -12385.331} C_VEL
LIN {X 0,Y 375.948,Z 165.656,A -85,B 0,C 180,E1 -12388.437,E2 -12388.437} C_VEL
LIN {X 0,Y 375.99,Z 165.652,A -85,B 0,C 180,E1 -12392.141,E2 -12392.141} C_VEL
LIN {X 0,Y 375.992,Z 165.648,A -85,B 0,C 180,E1 -12394.538,E2 -12394.538} C_VEL
LIN {X 0,Y 375.944,Z 165.656,A -85,B 0,C 180,E1 -12398.044,E2 -12398.044} C_VEL
LIN {X 0,Y 376.01,Z 165.65,A -85,B 0,C 180,E1 -12401.473,E2 -12401.473} C_VEL
LIN {X 0,Y 376.045,Z 165.642,A -85,B 0,C 180,E1 -12404.832,E2 -12404.832} C_VEL
LIN {X 0,Y 376.042,Z 165.642,A -85,B 0,C 180,E1 -12408.136,E2 -12408.136} C_VEL
LIN {X 0,Y 376.206,Z 165.622,A -85,B 0,C 180,E1 -12411.917,E2 -12411.917} C_VEL
LIN {X 0,Y 376.16,Z 165.629,A -85,B 0,C 180,E1 -12414.64,E2 -12414.64} C_VEL
LIN {X 0,Y 376.34,Z 165.605,A -85,B 0,C 180,E1 -12417.859,E2 -12417.859} C_VEL
LIN {X 0,Y 376.473,Z 165.588,A -85,B 0,C 180,E1 -12420,E2 -12420} C_VEL
LIN {X 0,Y 376.166,Z 165.628,A -85,B 0,C 180,E1 -12423.213,E2 -12423.213} C_VEL
LIN {X 0,Y 376.218,Z 165.621,A -85,B 0,C 180,E1 -12426.65,E2 -12426.65} C_VEL
LIN {X 0,Y 376.192,Z 165.627,A -85,B 0,C 180,E1 -12428.595,E2 -12428.595} C_VEL
LIN {X 0,Y 376.045,Z 165.642,A -85,B 0,C 180,E1 -12431.864,E2 -12431.864} C_VEL
LIN {X 0,Y 376.045,Z 165.641,A -85,B 0,C 180,E1 -12435.168,E2 -12435.168} C_VEL
LIN {X 0,Y 376.016,Z 165.648,A -85,B 0,C 180,E1 -12438.526,E2 -12438.526} C_VEL
LIN {X 0,Y 375.966,Z 165.655,A -85,B 0,C 180,E1 -12441.954,E2 -12441.954} C_VEL
LIN {X 0,Y 375.975,Z 165.654,A -85,B 0,C 180,E1 -12444.283,E2 -12444.283} C_VEL
LIN {X 0,Y 375.922,Z 165.66,A -85,B 0,C 180,E1 -12447.865,E2 -12447.865} C_VEL
LIN {X 0,Y 375.945,Z 165.656,A -85,B 0,C 180,E1 -12451.563,E2 -12451.563} C_VEL
LIN {X 0,Y 375.946,Z 165.656,A -85,B 0,C 180,E1 -12455.417,E2 -12455.417} C_VEL
LIN {X 0,Y 375.965,Z 165.652,A -85,B 0,C 180,E1 -12458.272,E2 -12458.272} C_VEL
LIN {X 0,Y 375.925,Z 165.661,A -85,B 0,C 180,E1 -12461.602,E2 -12461.602} C_VEL
LIN {X 0,Y 375.946,Z 165.658,A -85,B 0,C 180,E1 -12465.266,E2 -12465.266} C_VEL
LIN {X 0,Y 375.932,Z 165.658,A -85,B 0,C 180,E1 -12469.135,E2 -12469.135} C_VEL
LIN {X 0,Y 375.954,Z 165.653,A -85,B 0,C 180,E1 -12471.913,E2 -12471.913} C_VEL
LIN {X 0,Y 375.972,Z 165.653,A -85,B 0,C 180,E1 -12475.334,E2 -12475.334} C_VEL
LIN {X 0,Y 375.955,Z 165.654,A -85,B 0,C 180,E1 -12478.44,E2 -12478.44} C_VEL
LIN {X 0,Y 375.997,Z 165.648,A -85,B 0,C 180,E1 -12482.144,E2 -12482.144} C_VEL
LIN {X 0,Y 376,Z 165.649,A -85,B 0,C 180,E1 -12484.541,E2 -12484.541} C_VEL
LIN {X 0,Y 375.964,Z 165.652,A -85,B 0,C 180,E1 -12488.048,E2 -12488.048} C_VEL
LIN {X 0,Y 376.006,Z 165.647,A -85,B 0,C 180,E1 -12491.475,E2 -12491.475} C_VEL
LIN {X 0,Y 376.056,Z 165.643,A -85,B 0,C 180,E1 -12494.834,E2 -12494.834} C_VEL
LIN {X 0,Y 376.048,Z 165.643,A -85,B 0,C 180,E1 -12498.138,E2 -12498.138} C_VEL
LIN {X 0,Y 376.258,Z 165.617,A -85,B 0,C 180,E1 -12501.879,E2 -12501.879} C_VEL
LIN {X 0,Y 376.173,Z 165.628,A -85,B 0,C 180,E1 -12504.642,E2 -12504.642} C_VEL
LIN {X 0,Y 376.353,Z 165.606,A -85,B 0,C 180,E1 -12507.861,E2 -12507.861} C_VEL
LIN {X 0,Y 376.35,Z 165.606,A -85,B 0,C 180,E1 -12512.142,E2 -12512.142} C_VEL
LIN {X 0,Y 376.25,Z 165.617,A -85,B 0,C 180,E1 -12516.437,E2 -12516.437} C_VEL
LIN {X 0,Y 376.208,Z 165.621,A -85,B 0,C 180,E1 -12518.597,E2 -12518.597} C_VEL
LIN {X 0,Y 376.053,Z 165.643,A -85,B 0,C 180,E1 -12521.865,E2 -12521.865} C_VEL
LIN {X 0,Y 376.061,Z 165.642,A -85,B 0,C 180,E1 -12525.169,E2 -12525.169} C_VEL
LIN {X 0,Y 376.013,Z 165.646,A -85,B 0,C 180,E1 -12528.528,E2 -12528.528} C_VEL
LIN {X 0,Y 375.959,Z 165.653,A -85,B 0,C 180,E1 -12531.956,E2 -12531.956} C_VEL
LIN {X 0,Y 375.94,Z 165.654,A -85,B 0,C 180,E1 -12534.287,E2 -12534.287} C_VEL
LIN {X 0,Y 375.917,Z 165.658,A -85,B 0,C 180,E1 -12536.662,E2 -12536.662} C_VEL
LIN {X 0,Y 375.918,Z 165.661,A -85,B 0,C 180,E1 -12539.085,E2 -12539.085} C_VEL
LIN {X 0,Y 375.962,Z 165.653,A -85,B 0,C 180,E1 -12541.563,E2 -12541.563} C_VEL
LIN {X 0,Y 375.961,Z 165.653,A -85,B 0,C 180,E1 -12545.417,E2 -12545.417} C_VEL
LIN {X 0,Y 375.939,Z 165.656,A -85,B 0,C 180,E1 -12548.264,E2 -12548.264} C_VEL
LIN {X 0,Y 375.936,Z 165.654,A -85,B 0,C 180,E1 -12550.05,E2 -12550.05} C_VEL
LIN {X 0,Y 375.226,Z 165.746,A -85,B 0,C 180,E1 -12550.944,E2 -12550.944} C_VEL
LIN {X 0,Y 372.339,Z 166.107,A -85,B 0,C 180,E1 -12552.397,E2 -12552.397} C_VEL
LIN {X 0,Y 369.94,Z 166.402,A -85,B 0,C 180,E1 -12553.573,E2 -12553.573} C_VEL
LIN {X 0,Y 368.946,Z 166.529,A -85,B 0,C 180,E1 -12554.482,E2 -12554.482} C_VEL
LIN {X 0,Y 368.882,Z 166.536,A -85,B 0,C 180,E1 -12554.79,E2 -12554.79} C_VEL
LIN {X 0,Y 368.888,Z 166.536,A -85,B 0,C 180,E1 -12558.178,E2 -12558.178} C_VEL
LIN {X 0,Y 368.885,Z 166.532,A -85,B 0,C 180,E1 -12561.366,E2 -12561.366} C_VEL
LIN {X 0,Y 368.948,Z 166.527,A -85,B 0,C 180,E1 -12565.148,E2 -12565.148} C_VEL
LIN {X 0,Y 369.029,Z 166.724,A -85,B 0,C 180,E1 -12566.312,E2 -12566.312} C_VEL
LIN {X 0,Y 369.928,Z 172.457,A -85,B 0,C 180,E1 -12569.139,E2 -12569.139} C_VEL
LIN {X 0,Y 369.722,Z 177.722,A -85,B 0,C 180,E1 -12571.626,E2 -12571.626} C_VEL
LIN {X 0,Y 369.308,Z 184.248,A -85,B 0,C 180,E1 -12574.648,E2 -12574.648} C_VEL
LIN {X 0,Y 368.845,Z 192.027,A -85,B 0,C 180,E1 -12578.189,E2 -12578.189} C_VEL
LIN {X 0,Y 368.49,Z 199.768,A -85,B 0,C 180,E1 -12581.658,E2 -12581.658} C_VEL
LIN {X 0,Y 368.164,Z 207.464,A -85,B 0,C 180,E1 -12585.066,E2 -12585.066} C_VEL
LIN {X 0,Y 367.899,Z 215.152,A -85,B 0,C 180,E1 -12588.429,E2 -12588.429} C_VEL
LIN {X 0,Y 367.903,Z 215.91,A -85,B 0,C 180,E1 -12588.743,E2 -12588.743} C_VEL
LIN {X 0,Y 368.888,Z 227.414,A -85,B 0,C 180,E1 -12589.434,E2 -12589.434} C_VEL
LIN {X 0,Y 369.51,Z 234.687,A -85,B 0,C 180,E1 -12590.005,E2 -12590.005} C_VEL
LIN {X 0,Y 369.016,Z 244.555,A -85,B 0,C 180,E1 -12590.96,E2 -12590.96} C_VEL
LIN {X 0,Y 368.672,Z 253.346,A -85,B 0,C 180,E1 -12592.056,E2 -12592.056} C_VEL
LIN {X 0,Y 368.299,Z 260.51,A -85,B 0,C 180,E1 -12593.182,E2 -12593.182} C_VEL
LIN {X 0,Y 368.094,Z 267.239,A -85,B 0,C 180,E1 -12594.522,E2 -12594.522} C_VEL
LIN {X 0,Y 367.885,Z 271.587,A -85,B 0,C 180,E1 -12595.618,E2 -12595.618} C_VEL
LIN {X 0,Y 367.715,Z 276.499,A -85,B 0,C 180,E1 -12597.261,E2 -12597.261} C_VEL
LIN {X 0,Y 367.615,Z 279.707,A -85,B 0,C 180,E1 -12598.905,E2 -12598.905} C_VEL
LIN {X 0,Y 367.602,Z 280.981,A -85,B 0,C 180,E1 -12600,E2 -12600} C_VEL
LIN {X 0,Y 367.685,Z 281.586,A -85,B 0,C 180,E1 -12601.095,E2 -12601.095} C_VEL
LIN {X 0,Y 367.851,Z 281.531,A -85,B 0,C 180,E1 -12602.19,E2 -12602.19} C_VEL
LIN {X 0,Y 368.118,Z 280.822,A -85,B 0,C 180,E1 -12603.284,E2 -12603.284} C_VEL
LIN {X 0,Y 368.575,Z 279.447,A -85,B 0,C 180,E1 -12604.374,E2 -12604.374} C_VEL
LIN {X 0,Y 368.838,Z 276.175,A -85,B 0,C 180,E1 -12606.016,E2 -12606.016} C_VEL
LIN {X 0,Y 369.511,Z 271.214,A -85,B 0,C 180,E1 -12607.651,E2 -12607.651} C_VEL
LIN {X 0,Y 370.323,Z 265.84,A -85,B 0,C 180,E1 -12608.962,E2 -12608.962} C_VEL
LIN {X 0,Y 371.507,Z 258.126,A -85,B 0,C 180,E1 -12610.399,E2 -12610.399} C_VEL
LIN {X 0,Y 372.693,Z 249.146,A -85,B 0,C 180,E1 -12611.696,E2 -12611.696} C_VEL
LIN {X 0,Y 373.477,Z 241.011,A -85,B 0,C 180,E1 -12612.636,E2 -12612.636} C_VEL
LIN {X 0,Y 372.33,Z 231.096,A -85,B 0,C 180,E1 -12613.71,E2 -12613.71} C_VEL
LIN {X 0,Y 370.038,Z 220.58,A -85,B 0,C 180,E1 -12614.72,E2 -12614.72} C_VEL
LIN {X 0,Y 369.176,Z 217.292,A -85,B 0,C 180,E1 -12615.033,E2 -12615.033} C_VEL
LIN {X 0,Y 369.74,Z 211.13,A -85,B 0,C 180,E1 -12618.119,E2 -12618.119} C_VEL
LIN {X 0,Y 370.434,Z 204.486,A -85,B 0,C 180,E1 -12621.618,E2 -12621.618} C_VEL
LIN {X 0,Y 371.203,Z 199.034,A -85,B 0,C 180,E1 -12624.659,E2 -12624.659} C_VEL
LIN {X 0,Y 372.268,Z 193.22,A -85,B 0,C 180,E1 -12628.163,E2 -12628.163} C_VEL
LIN {X 0,Y 372.949,Z 189.594,A -85,B 0,C 180,E1 -12630.584,E2 -12630.584} C_VEL
LIN {X 0,Y 373.161,Z 187.635,A -85,B 0,C 180,E1 -12632.055,E2 -12632.055} C_VEL
LIN {X 0,Y 372.921,Z 185.025,A -85,B 0,C 180,E1 -12634.428,E2 -12634.428} C_VEL
LIN {X 0,Y 372.567,Z 182.314,A -85,B 0,C 180,E1 -12637.599,E2 -12637.599} C_VEL
LIN {X 0,Y 372.336,Z 180.938,A -85,B 0,C 180,E1 -12639.924,E2 -12639.924} C_VEL
LIN {X 0,Y 372.216,Z 180.019,A -85,B 0,C 180,E1 -12642.823,E2 -12642.823} C_VEL
LIN {X 0,Y 372.306,Z 180.057,A -85,B 0,C 180,E1 -12645.834,E2 -12645.834} C_VEL
LIN {X 0,Y 372.56,Z 181.088,A -85,B 0,C 180,E1 -12648.68,E2 -12648.68} C_VEL
LIN {X 0,Y 373.046,Z 183.11,A -85,B 0,C 180,E1 -12651.558,E2 -12651.558} C_VEL
LIN {X 0,Y 373.688,Z 186.023,A -85,B 0,C 180,E1 -12654.335,E2 -12654.335} C_VEL
LIN {X 0,Y 374.663,Z 190.586,A -85,B 0,C 180,E1 -12657.578,E2 -12657.578} C_VEL
LIN {X 0,Y 375.403,Z 195.358,A -85,B 0,C 180,E1 -12660.255,E2 -12660.255} C_VEL
LIN {X 0,Y 375.146,Z 198.497,A -85,B 0,C 180,E1 -12661.703,E2 -12661.703} C_VEL
LIN {X 0,Y 373.033,Z 206.952,A -85,B 0,C 180,E1 -12665.071,E2 -12665.071} C_VEL
LIN {X 0,Y 371.191,Z 217.608,A -85,B 0,C 180,E1 -12668.914,E2 -12668.914} C_VEL
LIN {X 0,Y 370.807,Z 220.575,A -85,B 0,C 180,E1 -12669.888,E2 -12669.888} C_VEL
LIN {X 0,Y 373.563,Z 233.142,A -85,B 0,C 180,E1 -12670.662,E2 -12670.662} C_VEL
LIN {X 0,Y 374.635,Z 242.828,A -85,B 0,C 180,E1 -12671.319,E2 -12671.319} C_VEL
LIN {X 0,Y 374.452,Z 251.593,A -85,B 0,C 180,E1 -12671.958,E2 -12671.958} C_VEL
LIN {X 0,Y 373.328,Z 262.663,A -85,B 0,C 180,E1 -12672.892,E2 -12672.892} C_VEL
LIN {X 0,Y 371.971,Z 273.856,A -85,B 0,C 180,E1 -12674.098,E2 -12674.098} C_VEL
LIN {X 0,Y 370.724,Z 283.339,A -85,B 0,C 180,E1 -12675.363,E2 -12675.363} C_VEL
LIN {X 0,Y 369.907,Z 292.06,A -85,B 0,C 180,E1 -12676.82,E2 -12676.82} C_VEL
LIN {X 0,Y 368.849,Z 300.089,A -85,B 0,C 180,E1 -12678.458,E2 -12678.458} C_VEL
LIN {X 0,Y 368.223,Z 306.543,A -85,B 0,C 180,E1 -12680.107,E2 -12680.107} C_VEL
LIN {X 0,Y 367.788,Z 311.639,A -85,B 0,C 180,E1 -12681.759,E2 -12681.759} C_VEL
LIN {X 0,Y 367.565,Z 315.584,A -85,B 0,C 180,E1 -12683.411,E2 -12683.411} C_VEL
LIN {X 0,Y 367.482,Z 317.622,A -85,B 0,C 180,E1 -12684.511,E2 -12684.511} C_VEL
LIN {X 0,Y 367.481,Z 319.223,A -85,B 0,C 180,E1 -12685.611,E2 -12685.611} C_VEL
LIN {X 0,Y 367.538,Z 321.069,A -85,B 0,C 180,E1 -12687.807,E2 -12687.807} C_VEL
LIN {X 0,Y 367.58,Z 321.373,A -85,B 0,C 180,E1 -12688.903,E2 -12688.903} C_VEL
LIN {X 0,Y 367.59,Z 321.203,A -85,B 0,C 180,E1 -12689.998,E2 -12689.998} C_VEL
LIN {X 0,Y 367.607,Z 320.621,A -85,B 0,C 180,E1 -12691.094,E2 -12691.094} C_VEL
LIN {X 0,Y 367.652,Z 319.618,A -85,B 0,C 180,E1 -12692.189,E2 -12692.189} C_VEL
LIN {X 0,Y 367.542,Z 318.104,A -85,B 0,C 180,E1 -12693.287,E2 -12693.287} C_VEL
LIN {X 0,Y 367.621,Z 314.988,A -85,B 0,C 180,E1 -12694.933,E2 -12694.933} C_VEL
LIN {X 0,Y 367.639,Z 310.7,A -85,B 0,C 180,E1 -12696.584,E2 -12696.584} C_VEL
LIN {X 0,Y 367.829,Z 305.138,A -85,B 0,C 180,E1 -12698.237,E2 -12698.237} C_VEL
LIN {X 0,Y 368.079,Z 298.001,A -85,B 0,C 180,E1 -12699.893,E2 -12699.893} C_VEL
LIN {X 0,Y 368.597,Z 289.036,A -85,B 0,C 180,E1 -12701.547,E2 -12701.547} C_VEL
LIN {X 0,Y 369.122,Z 279.625,A -85,B 0,C 180,E1 -12702.926,E2 -12702.926} C_VEL
LIN {X 0,Y 369.763,Z 268.599,A -85,B 0,C 180,E1 -12704.222,E2 -12704.222} C_VEL
LIN {X 0,Y 370.476,Z 257.304,A -85,B 0,C 180,E1 -12705.259,E2 -12705.259} C_VEL
LIN {X 0,Y 371.018,Z 245.792,A -85,B 0,C 180,E1 -12706.081,E2 -12706.081} C_VEL
LIN {X 0,Y 370.553,Z 238.092,A -85,B 0,C 180,E1 -12706.527,E2 -12706.527} C_VEL
LIN {X 0,Y 369.306,Z 225.167,A -85,B 0,C 180,E1 -12707.1,E2 -12707.1} C_VEL
LIN {X 0,Y 368.911,Z 220.225,A -85,B 0,C 180,E1 -12707.28,E2 -12707.28} C_VEL
LIN {X 0,Y 369.771,Z 209.393,A -85,B 0,C 180,E1 -12710.584,E2 -12710.584} C_VEL
LIN {X 0,Y 371.118,Z 196.319,A -85,B 0,C 180,E1 -12714.633,E2 -12714.633} C_VEL
LIN {X 0,Y 372.278,Z 186.471,A -85,B 0,C 180,E1 -12717.728,E2 -12717.728} C_VEL
LIN {X 0,Y 372.154,Z 183.25,A -85,B 0,C 180,E1 -12718.785,E2 -12718.785} C_VEL
LIN {X 0,Y 370.663,Z 175.525,A -85,B 0,C 180,E1 -12721.435,E2 -12721.435} C_VEL
LIN {X 0,Y 368.927,Z 166.534,A -85,B 0,C 180,E1 -12724.686,E2 -12724.686} C_VEL
LIN {X 0,Y 368.896,Z 166.532,A -85,B 0,C 180,E1 -12727.561,E2 -12727.561} C_VEL
LIN {X 0,Y 368.901,Z 166.534,A -85,B 0,C 180,E1 -12730.369,E2 -12730.369} C_VEL
LIN {X 0,Y 368.879,Z 166.533,A -85,B 0,C 180,E1 -12733.615,E2 -12733.615} C_VEL
LIN {X 0,Y 368.931,Z 166.531,A -85,B 0,C 180,E1 -12736.702,E2 -12736.702} C_VEL
LIN {X 0,Y 368.943,Z 166.527,A -85,B 0,C 180,E1 -12739.634,E2 -12739.634} C_VEL
LIN {X 0,Y 368.891,Z 166.532,A -85,B 0,C 180,E1 -12743.143,E2 -12743.143} C_VEL
LIN {X 0,Y 368.885,Z 166.535,A -85,B 0,C 180,E1 -12746.461,E2 -12746.461} C_VEL
LIN {X 0,Y 368.911,Z 166.533,A -85,B 0,C 180,E1 -12750.309,E2 -12750.309} C_VEL
LIN {X 0,Y 368.969,Z 166.526,A -85,B 0,C 180,E1 -12753.534,E2 -12753.534} C_VEL
LIN {X 0,Y 368.943,Z 166.526,A -85,B 0,C 180,E1 -12756.42,E2 -12756.42} C_VEL
LIN {X 0,Y 368.923,Z 166.531,A -85,B 0,C 180,E1 -12759.946,E2 -12759.946} C_VEL
LIN {X 0,Y 368.962,Z 166.527,A -85,B 0,C 180,E1 -12763.398,E2 -12763.398} C_VEL
LIN {X 0,Y 369.045,Z 166.514,A -85,B 0,C 180,E1 -12766.79,E2 -12766.79} C_VEL
LIN {X 0,Y 369.054,Z 166.511,A -85,B 0,C 180,E1 -12770.131,E2 -12770.131} C_VEL
LIN {X 0,Y 369.15,Z 166.5,A -85,B 0,C 180,E1 -12772.341,E2 -12772.341} C_VEL
LIN {X 0,Y 369.132,Z 166.503,A -85,B 0,C 180,E1 -12774.537,E2 -12774.537} C_VEL
LIN {X 0,Y 369.305,Z 166.481,A -85,B 0,C 180,E1 -12777.819,E2 -12777.819} C_VEL
LIN {X 0,Y 369.443,Z 166.463,A -85,B 0,C 180,E1 -12780,E2 -12780} C_VEL
LIN {X 0,Y 369.3,Z 166.481,A -85,B 0,C 180,E1 -12782.181,E2 -12782.181} C_VEL
LIN {X 0,Y 369.187,Z 166.499,A -85,B 0,C 180,E1 -12786.639,E2 -12786.639} C_VEL
LIN {X 0,Y 369.125,Z 166.507,A -85,B 0,C 180,E1 -12788.761,E2 -12788.761} C_VEL
LIN {X 0,Y 368.999,Z 166.521,A -85,B 0,C 180,E1 -12792.093,E2 -12792.093} C_VEL
LIN {X 0,Y 368.984,Z 166.52,A -85,B 0,C 180,E1 -12795.465,E2 -12795.465} C_VEL
LIN {X 0,Y 368.976,Z 166.523,A -85,B 0,C 180,E1 -12798.893,E2 -12798.893} C_VEL
LIN {X 0,Y 368.933,Z 166.531,A -85,B 0,C 180,E1 -12802.395,E2 -12802.395} C_VEL
LIN {X 0,Y 368.93,Z 166.531,A -85,B 0,C 180,E1 -12805.985,E2 -12805.985} C_VEL
LIN {X 0,Y 368.883,Z 166.536,A -85,B 0,C 180,E1 -12809.693,E2 -12809.693} C_VEL
LIN {X 0,Y 368.885,Z 166.533,A -85,B 0,C 180,E1 -12813.044,E2 -12813.044} C_VEL
LIN {X 0,Y 368.907,Z 166.533,A -85,B 0,C 180,E1 -12816.198,E2 -12816.198} C_VEL
LIN {X 0,Y 368.893,Z 166.532,A -85,B 0,C 180,E1 -12818.954,E2 -12818.954} C_VEL
LIN {X 0,Y 368.871,Z 166.537,A -85,B 0,C 180,E1 -12822.011,E2 -12822.011} C_VEL
LIN {X 0,Y 368.918,Z 166.532,A -85,B 0,C 180,E1 -12825.185,E2 -12825.185} C_VEL
LIN {X 0,Y 368.874,Z 166.535,A -85,B 0,C 180,E1 -12828.179,E2 -12828.179} C_VEL
LIN {X 0,Y 368.899,Z 166.536,A -85,B 0,C 180,E1 -12831.362,E2 -12831.362} C_VEL
LIN {X 0,Y 368.929,Z 166.532,A -85,B 0,C 180,E1 -12835.148,E2 -12835.148} C_VEL
LIN {X 0,Y 368.923,Z 166.532,A -85,B 0,C 180,E1 -12839.048,E2 -12839.048} C_VEL
LIN {X 0,Y 368.981,Z 166.522,A -85,B 0,C 180,E1 -12841.566,E2 -12841.566} C_VEL
LIN {X 0,Y 368.952,Z 166.526,A -85,B 0,C 180,E1 -12845.226,E2 -12845.226} C_VEL
LIN {X 0,Y 368.934,Z 166.53,A -85,B 0,C 180,E1 -12848.975,E2 -12848.975} C_VEL
LIN {X 0,Y 368.988,Z 166.523,A -85,B 0,C 180,E1 -12852.259,E2 -12852.259} C_VEL
LIN {X 0,Y 369.035,Z 166.517,A -85,B 0,C 180,E1 -12856.23,E2 -12856.23} C_VEL
LIN {X 0,Y 369.066,Z 166.514,A -85,B 0,C 180,E1 -12860.134,E2 -12860.134} C_VEL
LIN {X 0,Y 369.189,Z 166.499,A -85,B 0,C 180,E1 -12862.344,E2 -12862.344} C_VEL
LIN {X 0,Y 369.145,Z 166.504,A -85,B 0,C 180,E1 -12864.539,E2 -12864.539} C_VEL
LIN {X 0,Y 369.318,Z 166.482,A -85,B 0,C 180,E1 -12867.821,E2 -12867.821} C_VEL
LIN {X 0,Y 369.315,Z 166.482,A -85,B 0,C 180,E1 -12872.183,E2 -12872.183} C_VEL
LIN {X 0,Y 369.211,Z 166.493,A -85,B 0,C 180,E1 -12876.56,E2 -12876.56} C_VEL
LIN {X 0,Y 369.141,Z 166.501,A -85,B 0,C 180,E1 -12878.762,E2 -12878.762} C_VEL
LIN {X 0,Y 369.008,Z 166.519,A -85,B 0,C 180,E1 -12882.095,E2 -12882.095} C_VEL
LIN {X 0,Y 369,Z 166.523,A -85,B 0,C 180,E1 -12885.466,E2 -12885.466} C_VEL
LIN {X 0,Y 368.962,Z 166.525,A -85,B 0,C 180,E1 -12888.895,E2 -12888.895} C_VEL
LIN {X 0,Y 368.903,Z 166.531,A -85,B 0,C 180,E1 -12892.399,E2 -12892.399} C_VEL
LIN {X 0,Y 368.923,Z 166.527,A -85,B 0,C 180,E1 -12895.987,E2 -12895.987} C_VEL
LIN {X 0,Y 368.898,Z 166.532,A -85,B 0,C 180,E1 -12899.693,E2 -12899.693} C_VEL
LIN {X 0,Y 368.902,Z 166.535,A -85,B 0,C 180,E1 -12903.044,E2 -12903.044} C_VEL
LIN {X 0,Y 368.92,Z 166.53,A -85,B 0,C 180,E1 -12906.198,E2 -12906.198} C_VEL
LIN {X 0,Y 368.868,Z 166.535,A -85,B 0,C 180,E1 -12910.059,E2 -12910.059} C_VEL
LIN {X 0,Y 368.887,Z 166.533,A -85,B 0,C 180,E1 -12913.616,E2 -12913.616} C_VEL
LIN {X 0,Y 368.882,Z 166.536,A -85,B 0,C 180,E1 -12914.79,E2 -12914.79} C_VEL
LIN {X 0,Y 368.258,Z 166.62,A -85,B 0,C 180,E1 -12915.701,E2 -12915.701} C_VEL
LIN {X 0,Y 365.409,Z 166.973,A -85,B 0,C 180,E1 -12917.182,E2 -12917.182} C_VEL
LIN {X 0,Y 362.966,Z 167.275,A -85,B 0,C 180,E1 -12918.38,E2 -12918.38} C_VEL
LIN {X 0,Y 361.912,Z 167.401,A -85,B 0,C 180,E1 -12919.307,E2 -12919.307} C_VEL
LIN {X 0,Y 361.826,Z 167.412,A -85,B 0,C 180,E1 -12919.622,E2 -12919.622} C_VEL
LIN {X 0,Y 361.869,Z 167.407,A -85,B 0,C 180,E1 -12922.982,E2 -12922.982} C_VEL
LIN {X 0,Y 361.962,Z 167.507,A -85,B 0,C 180,E1 -12926.138,E2 -12926.138} C_VEL
LIN {X 0,Y 362.898,Z 173.465,A -85,B 0,C 180,E1 -12929.131,E2 -12929.131} C_VEL
LIN {X 0,Y 362.693,Z 178.743,A -85,B 0,C 180,E1 -12931.657,E2 -12931.657} C_VEL
LIN {X 0,Y 362.234,Z 185.308,A -85,B 0,C 180,E1 -12934.733,E2 -12934.733} C_VEL
LIN {X 0,Y 361.755,Z 193.096,A -85,B 0,C 180,E1 -12938.339,E2 -12938.339} C_VEL
LIN {X 0,Y 361.391,Z 200.835,A -85,B 0,C 180,E1 -12941.871,E2 -12941.871} C_VEL
LIN {X 0,Y 361.056,Z 208.563,A -85,B 0,C 180,E1 -12945.342,E2 -12945.342} C_VEL
LIN {X 0,Y 360.824,Z 215.891,A -85,B 0,C 180,E1 -12948.591,E2 -12948.591} C_VEL
LIN {X 0,Y 361.864,Z 228.141,A -85,B 0,C 180,E1 -12949.368,E2 -12949.368} C_VEL
LIN {X 0,Y 362.427,Z 235.301,A -85,B 0,C 180,E1 -12949.949,E2 -12949.949} C_VEL
LIN {X 0,Y 361.931,Z 245.056,A -85,B 0,C 180,E1 -12950.922,E2 -12950.922} C_VEL
LIN {X 0,Y 361.512,Z 254.742,A -85,B 0,C 180,E1 -12952.179,E2 -12952.179} C_VEL
LIN {X 0,Y 361.201,Z 261.517,A -85,B 0,C 180,E1 -12953.296,E2 -12953.296} C_VEL
LIN {X 0,Y 360.984,Z 268.237,A -85,B 0,C 180,E1 -12954.694,E2 -12954.694} C_VEL
LIN {X 0,Y 360.75,Z 273.38,A -85,B 0,C 180,E1 -12956.09,E2 -12956.09} C_VEL
LIN {X 0,Y 360.536,Z 277.847,A -85,B 0,C 180,E1 -12957.766,E2 -12957.766} C_VEL
LIN {X 0,Y 360.531,Z 279.902,A -85,B 0,C 180,E1 -12958.883,E2 -12958.883} C_VEL
LIN {X 0,Y 360.535,Z 281.273,A -85,B 0,C 180,E1 -12960,E2 -12960} C_VEL
LIN {X 0,Y 360.618,Z 281.98,A -85,B 0,C 180,E1 -12961.117,E2 -12961.117} C_VEL
LIN {X 0,Y 360.789,Z 282.031,A -85,B 0,C 180,E1 -12962.233,E2 -12962.233} C_VEL
LIN {X 0,Y 361.067,Z 281.432,A -85,B 0,C 180,E1 -12963.348,E2 -12963.348} C_VEL
LIN {X 0,Y 361.552,Z 280.167,A -85,B 0,C 180,E1 -12964.46,E2 -12964.46} C_VEL
LIN {X 0,Y 361.853,Z 277.078,A -85,B 0,C 180,E1 -12966.132,E2 -12966.132} C_VEL
LIN {X 0,Y 362.569,Z 272.33,A -85,B 0,C 180,E1 -12967.798,E2 -12967.798} C_VEL
LIN {X 0,Y 363.531,Z 266.517,A -85,B 0,C 180,E1 -12969.28,E2 -12969.28} C_VEL
LIN {X 0,Y 364.746,Z 259.318,A -85,B 0,C 180,E1 -12970.674,E2 -12970.674} C_VEL
LIN {X 0,Y 365.915,Z 251.183,A -85,B 0,C 180,E1 -12971.916,E2 -12971.916} C_VEL
LIN {X 0,Y 366.92,Z 243.443,A -85,B 0,C 180,E1 -12972.866,E2 -12972.866} C_VEL
LIN {X 0,Y 366.102,Z 234.577,A -85,B 0,C 180,E1 -12973.901,E2 -12973.901} C_VEL
LIN {X 0,Y 363.912,Z 223.434,A -85,B 0,C 180,E1 -12975.064,E2 -12975.064} C_VEL
LIN {X 0,Y 362.295,Z 217.424,A -85,B 0,C 180,E1 -12975.653,E2 -12975.653} C_VEL
LIN {X 0,Y 362.828,Z 212.201,A -85,B 0,C 180,E1 -12978.35,E2 -12978.35} C_VEL
LIN {X 0,Y 363.586,Z 205.641,A -85,B 0,C 180,E1 -12981.899,E2 -12981.899} C_VEL
LIN {X 0,Y 364.436,Z 200.107,A -85,B 0,C 180,E1 -12985.104,E2 -12985.104} C_VEL
LIN {X 0,Y 365.586,Z 194.374,A -85,B 0,C 180,E1 -12988.725,E2 -12988.725} C_VEL
LIN {X 0,Y 366.064,Z 192.192,A -85,B 0,C 180,E1 -12990.235,E2 -12990.235} C_VEL
LIN {X 0,Y 366.35,Z 189.315,A -85,B 0,C 180,E1 -12992.49,E2 -12992.49} C_VEL
LIN {X 0,Y 366.097,Z 186.623,A -85,B 0,C 180,E1 -12995.164,E2 -12995.164} C_VEL
LIN {X 0,Y 365.828,Z 184.417,A -85,B 0,C 180,E1 -12998.031,E2 -12998.031} C_VEL
LIN {X 0,Y 365.655,Z 183.053,A -85,B 0,C 180,E1 -13000.805,E2 -13000.805} C_VEL
LIN {X 0,Y 365.593,Z 182.474,A -85,B 0,C 180,E1 -13003.793,E2 -13003.793} C_VEL
LIN {X 0,Y 365.77,Z 182.899,A -85,B 0,C 180,E1 -13006.899,E2 -13006.899} C_VEL
LIN {X 0,Y 366.161,Z 184.568,A -85,B 0,C 180,E1 -13010.153,E2 -13010.153} C_VEL
LIN {X 0,Y 366.527,Z 186.204,A -85,B 0,C 180,E1 -13012.149,E2 -13012.149} C_VEL
LIN {X 0,Y 367.292,Z 189.813,A -85,B 0,C 180,E1 -13015.365,E2 -13015.365} C_VEL
LIN {X 0,Y 367.993,Z 193.113,A -85,B 0,C 180,E1 -13017.671,E2 -13017.671} C_VEL
LIN {X 0,Y 368.661,Z 197.694,A -85,B 0,C 180,E1 -13020.286,E2 -13020.286} C_VEL
LIN {X 0,Y 368.378,Z 200.25,A -85,B 0,C 180,E1 -13021.512,E2 -13021.512} C_VEL
LIN {X 0,Y 366.143,Z 208.855,A -85,B 0,C 180,E1 -13025.02,E2 -13025.02} C_VEL
LIN {X 0,Y 364.388,Z 218.185,A -85,B 0,C 180,E1 -13028.501,E2 -13028.501} C_VEL
LIN {X 0,Y 364.095,Z 220.647,A -85,B 0,C 180,E1 -13029.298,E2 -13029.298} C_VEL
LIN {X 0,Y 366.84,Z 232.82,A -85,B 0,C 180,E1 -13030.099,E2 -13030.099} C_VEL
LIN {X 0,Y 368.164,Z 243.831,A -85,B 0,C 180,E1 -13030.895,E2 -13030.895} C_VEL
LIN {X 0,Y 367.833,Z 253.297,A -85,B 0,C 180,E1 -13031.622,E2 -13031.622} C_VEL
LIN {X 0,Y 366.455,Z 265.149,A -85,B 0,C 180,E1 -13032.705,E2 -13032.705} C_VEL
LIN {X 0,Y 365.01,Z 275.776,A -85,B 0,C 180,E1 -13033.93,E2 -13033.93} C_VEL
LIN {X 0,Y 363.626,Z 286.174,A -85,B 0,C 180,E1 -13035.446,E2 -13035.446} C_VEL
LIN {X 0,Y 362.827,Z 293.874,A -85,B 0,C 180,E1 -13036.843,E2 -13036.843} C_VEL
LIN {X 0,Y 361.729,Z 301.427,A -85,B 0,C 180,E1 -13038.511,E2 -13038.511} C_VEL
LIN {X 0,Y 361.009,Z 308.401,A -85,B 0,C 180,E1 -13040.474,E2 -13040.474} C_VEL
LIN {X 0,Y 360.645,Z 312.998,A -85,B 0,C 180,E1 -13042.158,E2 -13042.158} C_VEL
LIN {X 0,Y 360.442,Z 316.646,A -85,B 0,C 180,E1 -13043.942,E2 -13043.942} C_VEL
LIN {X 0,Y 360.388,Z 318.934,A -85,B 0,C 180,E1 -13045.524,E2 -13045.524} C_VEL
LIN {X 0,Y 360.439,Z 320.7,A -85,B 0,C 180,E1 -13047.763,E2 -13047.763} C_VEL
LIN {X 0,Y 360.515,Z 320.926,A -85,B 0,C 180,E1 -13048.881,E2 -13048.881} C_VEL
LIN {X 0,Y 360.523,Z 320.713,A -85,B 0,C 180,E1 -13049.998,E2 -13049.998} C_VEL
LIN {X 0,Y 360.542,Z 320.093,A -85,B 0,C 180,E1 -13051.115,E2 -13051.115} C_VEL
LIN {X 0,Y 360.587,Z 319.006,A -85,B 0,C 180,E1 -13052.232,E2 -13052.232} C_VEL
LIN {X 0,Y 360.454,Z 316.499,A -85,B 0,C 180,E1 -13053.911,E2 -13053.911} C_VEL
LIN {X 0,Y 360.511,Z 312.891,A -85,B 0,C 180,E1 -13055.592,E2 -13055.592} C_VEL
LIN {X 0,Y 360.602,Z 308.066,A -85,B 0,C 180,E1 -13057.276,E2 -13057.276} C_VEL
LIN {X 0,Y 360.801,Z 301.874,A -85,B 0,C 180,E1 -13058.963,E2 -13058.963} C_VEL
LIN {X 0,Y 361.155,Z 293.969,A -85,B 0,C 180,E1 -13060.651,E2 -13060.651} C_VEL
LIN {X 0,Y 361.68,Z 285.84,A -85,B 0,C 180,E1 -13062.055,E2 -13062.055} C_VEL
LIN {X 0,Y 362.339,Z 275.79,A -85,B 0,C 180,E1 -13063.457,E2 -13063.457} C_VEL
LIN {X 0,Y 362.843,Z 265.74,A -85,B 0,C 180,E1 -13064.582,E2 -13064.582} C_VEL
LIN {X 0,Y 363.546,Z 254.854,A -85,B 0,C 180,E1 -13065.557,E2 -13065.557} C_VEL
LIN {X 0,Y 363.999,Z 243.749,A -85,B 0,C 180,E1 -13066.328,E2 -13066.328} C_VEL
LIN {X 0,Y 362.708,Z 230.661,A -85,B 0,C 180,E1 -13067.025,E2 -13067.025} C_VEL
LIN {X 0,Y 361.858,Z 220.206,A -85,B 0,C 180,E1 -13067.426,E2 -13067.426} C_VEL
LIN {X 0,Y 362.813,Z 208.811,A -85,B 0,C 180,E1 -13070.997,E2 -13070.997} C_VEL
LIN {X 0,Y 364.149,Z 196.524,A -85,B 0,C 180,E1 -13074.893,E2 -13074.893} C_VEL
LIN {X 0,Y 365.244,Z 187.671,A -85,B 0,C 180,E1 -13077.732,E2 -13077.732} C_VEL
LIN {X 0,Y 365.189,Z 184.576,A -85,B 0,C 180,E1 -13078.756,E2 -13078.756} C_VEL
LIN {X 0,Y 363.538,Z 176.146,A -85,B 0,C 180,E1 -13081.721,E2 -13081.721} C_VEL
LIN {X 0,Y 361.901,Z 167.409,A -85,B 0,C 180,E1 -13084.949,E2 -13084.949} C_VEL
LIN {X 0,Y 361.86,Z 167.411,A -85,B 0,C 180,E1 -13088.423,E2 -13088.423} C_VEL
LIN {X 0,Y 361.817,Z 167.413,A -85,B 0,C 180,E1 -13091.329,E2 -13091.329} C_VEL
LIN {X 0,Y 361.837,Z 167.415,A -85,B 0,C 180,E1 -13094.362,E2 -13094.362} C_VEL
LIN {X 0,Y 361.875,Z 167.406,A -85,B 0,C 180,E1 -13097.558,E2 -13097.558} C_VEL
LIN {X 0,Y 361.863,Z 167.408,A -85,B 0,C 180,E1 -13100.971,E2 -13100.971} C_VEL
LIN {X 0,Y 361.863,Z 167.409,A -85,B 0,C 180,E1 -13104.654,E2 -13104.654} C_VEL
LIN {X 0,Y 361.826,Z 167.415,A -85,B 0,C 180,E1 -13108.369,E2 -13108.369} C_VEL
LIN {X 0,Y 361.89,Z 167.404,A -85,B 0,C 180,E1 -13110.954,E2 -13110.954} C_VEL
LIN {X 0,Y 361.942,Z 167.4,A -85,B 0,C 180,E1 -13113.474,E2 -13113.474} C_VEL
LIN {X 0,Y 361.869,Z 167.407,A -85,B 0,C 180,E1 -13117.143,E2 -13117.143} C_VEL
LIN {X 0,Y 361.907,Z 167.402,A -85,B 0,C 180,E1 -13120.723,E2 -13120.723} C_VEL
LIN {X 0,Y 361.932,Z 167.4,A -85,B 0,C 180,E1 -13124.225,E2 -13124.225} C_VEL
LIN {X 0,Y 361.986,Z 167.392,A -85,B 0,C 180,E1 -13126.527,E2 -13126.527} C_VEL
LIN {X 0,Y 362.018,Z 167.389,A -85,B 0,C 180,E1 -13129.937,E2 -13129.937} C_VEL
LIN {X 0,Y 362.151,Z 167.376,A -85,B 0,C 180,E1 -13133.313,E2 -13133.313} C_VEL
LIN {X 0,Y 362.269,Z 167.358,A -85,B 0,C 180,E1 -13137.776,E2 -13137.776} C_VEL
LIN {X 0,Y 362.412,Z 167.339,A -85,B 0,C 180,E1 -13140,E2 -13140} C_VEL
LIN {X 0,Y 362.264,Z 167.358,A -85,B 0,C 180,E1 -13142.224,E2 -13142.224} C_VEL
LIN {X 0,Y 362.157,Z 167.376,A -85,B 0,C 180,E1 -13146.686,E2 -13146.686} C_VEL
LIN {X 0,Y 362.061,Z 167.387,A -85,B 0,C 180,E1 -13148.933,E2 -13148.933} C_VEL
LIN {X 0,Y 361.953,Z 167.4,A -85,B 0,C 180,E1 -13152.333,E2 -13152.333} C_VEL
LIN {X 0,Y 361.948,Z 167.401,A -85,B 0,C 180,E1 -13154.621,E2 -13154.621} C_VEL
LIN {X 0,Y 361.947,Z 167.4,A -85,B 0,C 180,E1 -13158.1,E2 -13158.1} C_VEL
LIN {X 0,Y 361.889,Z 167.405,A -85,B 0,C 180,E1 -13161.653,E2 -13161.653} C_VEL
LIN {X 0,Y 361.883,Z 167.405,A -85,B 0,C 180,E1 -13165.293,E2 -13165.293} C_VEL
LIN {X 0,Y 361.842,Z 167.41,A -85,B 0,C 180,E1 -13169.075,E2 -13169.075} C_VEL
LIN {X 0,Y 361.836,Z 167.411,A -85,B 0,C 180,E1 -13172.946,E2 -13172.946} C_VEL
LIN {X 0,Y 361.857,Z 167.412,A -85,B 0,C 180,E1 -13175.638,E2 -13175.638} C_VEL
LIN {X 0,Y 361.86,Z 167.408,A -85,B 0,C 180,E1 -13179.028,E2 -13179.028} C_VEL
LIN {X 0,Y 361.827,Z 167.412,A -85,B 0,C 180,E1 -13182.83,E2 -13182.83} C_VEL
LIN {X 0,Y 361.827,Z 167.414,A -85,B 0,C 180,E1 -13185.945,E2 -13185.945} C_VEL
LIN {X 0,Y 361.827,Z 167.416,A -85,B 0,C 180,E1 -13189.246,E2 -13189.246} C_VEL
LIN {X 0,Y 361.855,Z 167.41,A -85,B 0,C 180,E1 -13192.779,E2 -13192.779} C_VEL
LIN {X 0,Y 361.847,Z 167.411,A -85,B 0,C 180,E1 -13195.721,E2 -13195.721} C_VEL
LIN {X 0,Y 361.871,Z 167.408,A -85,B 0,C 180,E1 -13199.674,E2 -13199.674} C_VEL
LIN {X 0,Y 361.949,Z 167.398,A -85,B 0,C 180,E1 -13203.477,E2 -13203.477} C_VEL
LIN {X 0,Y 361.887,Z 167.407,A -85,B 0,C 180,E1 -13207.147,E2 -13207.147} C_VEL
LIN {X 0,Y 361.904,Z 167.406,A -85,B 0,C 180,E1 -13210.725,E2 -13210.725} C_VEL
LIN {X 0,Y 361.93,Z 167.401,A -85,B 0,C 180,E1 -13213.068,E2 -13213.068} C_VEL
LIN {X 0,Y 361.998,Z 167.396,A -85,B 0,C 180,E1 -13216.53,E2 -13216.53} C_VEL
LIN {X 0,Y 362.03,Z 167.389,A -85,B 0,C 180,E1 -13219.94,E2 -13219.94} C_VEL
LIN {X 0,Y 362.152,Z 167.376,A -85,B 0,C 180,E1 -13222.194,E2 -13222.194} C_VEL
LIN {X 0,Y 362.119,Z 167.38,A -85,B 0,C 180,E1 -13224.433,E2 -13224.433} C_VEL
LIN {X 0,Y 362.282,Z 167.359,A -85,B 0,C 180,E1 -13227.778,E2 -13227.778} C_VEL
LIN {X 0,Y 362.279,Z 167.358,A -85,B 0,C 180,E1 -13232.225,E2 -13232.225} C_VEL
LIN {X 0,Y 362.175,Z 167.369,A -85,B 0,C 180,E1 -13236.688,E2 -13236.688} C_VEL
LIN {X 0,Y 362.077,Z 167.381,A -85,B 0,C 180,E1 -13238.935,E2 -13238.935} C_VEL
LIN {X 0,Y 361.963,Z 167.395,A -85,B 0,C 180,E1 -13242.334,E2 -13242.334} C_VEL
LIN {X 0,Y 361.965,Z 167.394,A -85,B 0,C 180,E1 -13244.622,E2 -13244.622} C_VEL
LIN {X 0,Y 361.96,Z 167.396,A -85,B 0,C 180,E1 -13248.101,E2 -13248.101} C_VEL
LIN {X 0,Y 361.858,Z 167.411,A -85,B 0,C 180,E1 -13251.657,E2 -13251.657} C_VEL
LIN {X 0,Y 361.864,Z 167.411,A -85,B 0,C 180,E1 -13255.296,E2 -13255.296} C_VEL
LIN {X 0,Y 361.86,Z 167.412,A -85,B 0,C 180,E1 -13259.075,E2 -13259.075} C_VEL
LIN {X 0,Y 361.853,Z 167.413,A -85,B 0,C 180,E1 -13262.946,E2 -13262.946} C_VEL
LIN {X 0,Y 361.872,Z 167.407,A -85,B 0,C 180,E1 -13265.638,E2 -13265.638} C_VEL
LIN {X 0,Y 361.83,Z 167.414,A -85,B 0,C 180,E1 -13269.019,E2 -13269.019} C_VEL
LIN {X 0,Y 361.838,Z 167.414,A -85,B 0,C 180,E1 -13272.83,E2 -13272.83} C_VEL
LIN {X 0,Y 361.823,Z 167.414,A -85,B 0,C 180,E1 -13275.948,E2 -13275.948} C_VEL
LIN {X 0,Y 361.839,Z 167.41,A -85,B 0,C 180,E1 -13279.246,E2 -13279.246} C_VEL
LIN {X 0,Y 361.826,Z 167.412,A -85,B 0,C 180,E1 -13279.622,E2 -13279.622} C_VEL
LIN {X 0,Y 361.161,Z 167.499,A -85,B 0,C 180,E1 -13280.55,E2 -13280.55} C_VEL
LIN {X 0,Y 358.324,Z 167.856,A -85,B 0,C 180,E1 -13282.061,E2 -13282.061} C_VEL
LIN {X 0,Y 355.928,Z 168.154,A -85,B 0,C 180,E1 -13283.284,E2 -13283.284} C_VEL
LIN {X 0,Y 354.906,Z 168.279,A -85,B 0,C 180,E1 -13284.229,E2 -13284.229} C_VEL
LIN {X 0,Y 354.827,Z 168.286,A -85,B 0,C 180,E1 -13284.549,E2 -13284.549} C_VEL
LIN {X 0,Y 354.915,Z 168.313,A -85,B 0,C 180,E1 -13285.986,E2 -13285.986} C_VEL
LIN {X 0,Y 355.883,Z 174.435,A -85,B 0,C 180,E1 -13289.106,E2 -13289.106} C_VEL
LIN {X 0,Y 355.661,Z 179.742,A -85,B 0,C 180,E1 -13291.69,E2 -13291.69} C_VEL
LIN {X 0,Y 355.168,Z 186.306,A -85,B 0,C 180,E1 -13294.822,E2 -13294.822} C_VEL
LIN {X 0,Y 354.675,Z 194.455,A -85,B 0,C 180,E1 -13298.645,E2 -13298.645} C_VEL
LIN {X 0,Y 354.28,Z 202.178,A -85,B 0,C 180,E1 -13302.216,E2 -13302.216} C_VEL
LIN {X 0,Y 353.915,Z 210.947,A -85,B 0,C 180,E1 -13306.214,E2 -13306.214} C_VEL
LIN {X 0,Y 353.737,Z 215.933,A -85,B 0,C 180,E1 -13308.468,E2 -13308.468} C_VEL
LIN {X 0,Y 354.81,Z 228.692,A -85,B 0,C 180,E1 -13309.298,E2 -13309.298} C_VEL
LIN {X 0,Y 355.337,Z 235.775,A -85,B 0,C 180,E1 -13309.89,E2 -13309.89} C_VEL
LIN {X 0,Y 354.839,Z 245.474,A -85,B 0,C 180,E1 -13310.883,E2 -13310.883} C_VEL
LIN {X 0,Y 354.46,Z 254.168,A -85,B 0,C 180,E1 -13312.022,E2 -13312.022} C_VEL
LIN {X 0,Y 354.073,Z 262.634,A -85,B 0,C 180,E1 -13313.447,E2 -13313.447} C_VEL
LIN {X 0,Y 353.863,Z 269.177,A -85,B 0,C 180,E1 -13314.873,E2 -13314.873} C_VEL
LIN {X 0,Y 353.563,Z 275.03,A -85,B 0,C 180,E1 -13316.581,E2 -13316.581} C_VEL
LIN {X 0,Y 353.454,Z 279.089,A -85,B 0,C 180,E1 -13318.291,E2 -13318.291} C_VEL
LIN {X 0,Y 353.469,Z 281.554,A -85,B 0,C 180,E1 -13320,E2 -13320} C_VEL
LIN {X 0,Y 353.554,Z 282.371,A -85,B 0,C 180,E1 -13321.139,E2 -13321.139} C_VEL
LIN {X 0,Y 353.731,Z 282.535,A -85,B 0,C 180,E1 -13322.277,E2 -13322.277} C_VEL
LIN {X 0,Y 354.019,Z 282.043,A -85,B 0,C 180,E1 -13323.414,E2 -13323.414} C_VEL
LIN {X 0,Y 354.527,Z 280.886,A -85,B 0,C 180,E1 -13324.548,E2 -13324.548} C_VEL
LIN {X 0,Y 354.851,Z 277.971,A -85,B 0,C 180,E1 -13326.254,E2 -13326.254} C_VEL
LIN {X 0,Y 355.631,Z 273.454,A -85,B 0,C 180,E1 -13327.952,E2 -13327.952} C_VEL
LIN {X 0,Y 356.806,Z 267.107,A -85,B 0,C 180,E1 -13329.64,E2 -13329.64} C_VEL
LIN {X 0,Y 357.938,Z 260.984,A -85,B 0,C 180,E1 -13330.88,E2 -13330.88} C_VEL
LIN {X 0,Y 359.153,Z 253.22,A -85,B 0,C 180,E1 -13332.144,E2 -13332.144} C_VEL
LIN {X 0,Y 360.361,Z 244.732,A -85,B 0,C 180,E1 -13333.248,E2 -13333.248} C_VEL
LIN {X 0,Y 359.51,Z 235.179,A -85,B 0,C 180,E1 -13334.421,E2 -13334.421} C_VEL
LIN {X 0,Y 357.472,Z 224.964,A -85,B 0,C 180,E1 -13335.555,E2 -13335.555} C_VEL
LIN {X 0,Y 355.446,Z 217.501,A -85,B 0,C 180,E1 -13336.365,E2 -13336.365} C_VEL
LIN {X 0,Y 356.117,Z 211.474,A -85,B 0,C 180,E1 -13339.603,E2 -13339.603} C_VEL
LIN {X 0,Y 357,Z 205.17,A -85,B 0,C 180,E1 -13343.187,E2 -13343.187} C_VEL
LIN {X 0,Y 358.069,Z 199.259,A -85,B 0,C 180,E1 -13346.836,E2 -13346.836} C_VEL
LIN {X 0,Y 358.944,Z 195.597,A -85,B 0,C 180,E1 -13349.307,E2 -13349.307} C_VEL
LIN {X 0,Y 359.525,Z 192.269,A -85,B 0,C 180,E1 -13351.857,E2 -13351.857} C_VEL
LIN {X 0,Y 359.559,Z 190.803,A -85,B 0,C 180,E1 -13353.182,E2 -13353.182} C_VEL
LIN {X 0,Y 359.331,Z 188.296,A -85,B 0,C 180,E1 -13355.927,E2 -13355.927} C_VEL
LIN {X 0,Y 359.088,Z 186.444,A -85,B 0,C 180,E1 -13358.778,E2 -13358.778} C_VEL
LIN {X 0,Y 358.954,Z 185.271,A -85,B 0,C 180,E1 -13361.924,E2 -13361.924} C_VEL
LIN {X 0,Y 359.03,Z 185.113,A -85,B 0,C 180,E1 -13365.193,E2 -13365.193} C_VEL
LIN {X 0,Y 359.313,Z 186.05,A -85,B 0,C 180,E1 -13368.314,E2 -13368.314} C_VEL
LIN {X 0,Y 359.747,Z 188.072,A -85,B 0,C 180,E1 -13371.393,E2 -13371.393} C_VEL
LIN {X 0,Y 360.305,Z 190.85,A -85,B 0,C 180,E1 -13374.183,E2 -13374.183} C_VEL
LIN {X 0,Y 361.112,Z 194.484,A -85,B 0,C 180,E1 -13376.978,E2 -13376.978} C_VEL
LIN {X 0,Y 361.801,Z 198.799,A -85,B 0,C 180,E1 -13379.664,E2 -13379.664} C_VEL
LIN {X 0,Y 361.759,Z 201.298,A -85,B 0,C 180,E1 -13380.954,E2 -13380.954} C_VEL
LIN {X 0,Y 360.285,Z 206.767,A -85,B 0,C 180,E1 -13383.341,E2 -13383.341} C_VEL
LIN {X 0,Y 357.905,Z 217.399,A -85,B 0,C 180,E1 -13387.53,E2 -13387.53} C_VEL
LIN {X 0,Y 357.362,Z 220.406,A -85,B 0,C 180,E1 -13388.644,E2 -13388.644} C_VEL
LIN {X 0,Y 360.4,Z 233.305,A -85,B 0,C 180,E1 -13389.559,E2 -13389.559} C_VEL
LIN {X 0,Y 361.71,Z 244.565,A -85,B 0,C 180,E1 -13390.426,E2 -13390.426} C_VEL
LIN {X 0,Y 361.419,Z 253.382,A -85,B 0,C 180,E1 -13391.137,E2 -13391.137} C_VEL
LIN {X 0,Y 359.955,Z 265.077,A -85,B 0,C 180,E1 -13392.236,E2 -13392.236} C_VEL
LIN {X 0,Y 358.463,Z 275.592,A -85,B 0,C 180,E1 -13393.482,E2 -13393.482} C_VEL
LIN {X 0,Y 356.974,Z 285.231,A -85,B 0,C 180,E1 -13394.906,E2 -13394.906} C_VEL
LIN {X 0,Y 355.925,Z 294.242,A -85,B 0,C 180,E1 -13396.583,E2 -13396.583} C_VEL
LIN {X 0,Y 354.774,Z 301.631,A -85,B 0,C 180,E1 -13398.283,E2 -13398.283} C_VEL
LIN {X 0,Y 353.982,Z 308.426,A -85,B 0,C 180,E1 -13400.283,E2 -13400.283} C_VEL
LIN {X 0,Y 353.589,Z 312.909,A -85,B 0,C 180,E1 -13402.001,E2 -13402.001} C_VEL
LIN {X 0,Y 353.335,Z 316.755,A -85,B 0,C 180,E1 -13404.002,E2 -13404.002} C_VEL
LIN {X 0,Y 353.299,Z 318.655,A -85,B 0,C 180,E1 -13405.434,E2 -13405.434} C_VEL
LIN {X 0,Y 353.277,Z 319.695,A -85,B 0,C 180,E1 -13406.577,E2 -13406.577} C_VEL
LIN {X 0,Y 353.341,Z 320.313,A -85,B 0,C 180,E1 -13407.718,E2 -13407.718} C_VEL
LIN {X 0,Y 353.45,Z 320.472,A -85,B 0,C 180,E1 -13408.859,E2 -13408.859} C_VEL
LIN {X 0,Y 353.458,Z 320.218,A -85,B 0,C 180,E1 -13409.998,E2 -13409.998} C_VEL
LIN {X 0,Y 353.48,Z 319.535,A -85,B 0,C 180,E1 -13411.137,E2 -13411.137} C_VEL
LIN {X 0,Y 353.523,Z 318.372,A -85,B 0,C 180,E1 -13412.277,E2 -13412.277} C_VEL
LIN {X 0,Y 353.382,Z 315.764,A -85,B 0,C 180,E1 -13413.99,E2 -13413.99} C_VEL
LIN {X 0,Y 353.454,Z 312.053,A -85,B 0,C 180,E1 -13415.704,E2 -13415.704} C_VEL
LIN {X 0,Y 353.559,Z 307.114,A -85,B 0,C 180,E1 -13417.422,E2 -13417.422} C_VEL
LIN {X 0,Y 353.755,Z 300.736,A -85,B 0,C 180,E1 -13419.143,E2 -13419.143} C_VEL
LIN {X 0,Y 354.12,Z 292.655,A -85,B 0,C 180,E1 -13420.866,E2 -13420.866} C_VEL
LIN {X 0,Y 354.643,Z 284.327,A -85,B 0,C 180,E1 -13422.298,E2 -13422.298} C_VEL
LIN {X 0,Y 355.313,Z 273.937,A -85,B 0,C 180,E1 -13423.729,E2 -13423.729} C_VEL
LIN {X 0,Y 355.893,Z 263.601,A -85,B 0,C 180,E1 -13424.873,E2 -13424.873} C_VEL
LIN {X 0,Y 356.642,Z 252.132,A -85,B 0,C 180,E1 -13425.866,E2 -13425.866} C_VEL
LIN {X 0,Y 356.906,Z 243.882,A -85,B 0,C 180,E1 -13426.441,E2 -13426.441} C_VEL
LIN {X 0,Y 355.533,Z 230.101,A -85,B 0,C 180,E1 -13427.191,E2 -13427.191} C_VEL
LIN {X 0,Y 354.807,Z 220.181,A -85,B 0,C 180,E1 -13427.581,E2 -13427.581} C_VEL
LIN {X 0,Y 355.824,Z 208.363,A -85,B 0,C 180,E1 -13431.37,E2 -13431.37} C_VEL
LIN {X 0,Y 357.18,Z 196.674,A -85,B 0,C 180,E1 -13435.161,E2 -13435.161} C_VEL
LIN {X 0,Y 358.286,Z 187.814,A -85,B 0,C 180,E1 -13438.082,E2 -13438.082} C_VEL
LIN {X 0,Y 357.719,Z 183.011,A -85,B 0,C 180,E1 -13439.756,E2 -13439.756} C_VEL
LIN {X 0,Y 355.485,Z 171.727,A -85,B 0,C 180,E1 -13443.865,E2 -13443.865} C_VEL
LIN {X 0,Y 354.835,Z 168.29,A -85,B 0,C 180,E1 -13445.214,E2 -13445.214} C_VEL
LIN {X 0,Y 354.798,Z 168.288,A -85,B 0,C 180,E1 -13447.881,E2 -13447.881} C_VEL
LIN {X 0,Y 354.778,Z 168.291,A -85,B 0,C 180,E1 -13451.169,E2 -13451.169} C_VEL
LIN {X 0,Y 354.806,Z 168.291,A -85,B 0,C 180,E1 -13454.513,E2 -13454.513} C_VEL
LIN {X 0,Y 354.828,Z 168.284,A -85,B 0,C 180,E1 -13457.667,E2 -13457.667} C_VEL
LIN {X 0,Y 354.812,Z 168.288,A -85,B 0,C 180,E1 -13460.665,E2 -13460.665} C_VEL
LIN {X 0,Y 354.811,Z 168.29,A -85,B 0,C 180,E1 -13464.299,E2 -13464.299} C_VEL
LIN {X 0,Y 354.775,Z 168.292,A -85,B 0,C 180,E1 -13467.665,E2 -13467.665} C_VEL
LIN {X 0,Y 354.857,Z 168.281,A -85,B 0,C 180,E1 -13470.62,E2 -13470.62} C_VEL
LIN {X 0,Y 354.886,Z 168.279,A -85,B 0,C 180,E1 -13474.171,E2 -13474.171} C_VEL
LIN {X 0,Y 354.803,Z 168.291,A -85,B 0,C 180,E1 -13477.892,E2 -13477.892} C_VEL
LIN {X 0,Y 354.909,Z 168.277,A -85,B 0,C 180,E1 -13481.89,E2 -13481.89} C_VEL
LIN {X 0,Y 354.929,Z 168.273,A -85,B 0,C 180,E1 -13485.98,E2 -13485.98} C_VEL
LIN {X 0,Y 354.965,Z 168.268,A -85,B 0,C 180,E1 -13489.735,E2 -13489.735} C_VEL
LIN {X 0,Y 355.115,Z 168.253,A -85,B 0,C 180,E1 -13493.18,E2 -13493.18} C_VEL
LIN {X 0,Y 355.232,Z 168.234,A -85,B 0,C 180,E1 -13497.732,E2 -13497.732} C_VEL
LIN {X 0,Y 355.382,Z 168.215,A -85,B 0,C 180,E1 -13500,E2 -13500} C_VEL
LIN {X 0,Y 355.227,Z 168.234,A -85,B 0,C 180,E1 -13502.268,E2 -13502.268} C_VEL
LIN {X 0,Y 355.123,Z 168.251,A -85,B 0,C 180,E1 -13506.819,E2 -13506.819} C_VEL
LIN {X 0,Y 355.002,Z 168.264,A -85,B 0,C 180,E1 -13509.113,E2 -13509.113} C_VEL
LIN {X 0,Y 354.912,Z 168.278,A -85,B 0,C 180,E1 -13512.581,E2 -13512.581} C_VEL
LIN {X 0,Y 354.876,Z 168.28,A -85,B 0,C 180,E1 -13516.097,E2 -13516.097} C_VEL
LIN {X 0,Y 354.895,Z 168.28,A -85,B 0,C 180,E1 -13518.472,E2 -13518.472} C_VEL
LIN {X 0,Y 354.83,Z 168.288,A -85,B 0,C 180,E1 -13522.106,E2 -13522.106} C_VEL
LIN {X 0,Y 354.839,Z 168.285,A -85,B 0,C 180,E1 -13525.832,E2 -13525.832} C_VEL
LIN {X 0,Y 354.786,Z 168.291,A -85,B 0,C 180,E1 -13529.685,E2 -13529.685} C_VEL
LIN {X 0,Y 354.774,Z 168.293,A -85,B 0,C 180,E1 -13532.335,E2 -13532.335} C_VEL
LIN {X 0,Y 354.811,Z 168.29,A -85,B 0,C 180,E1 -13535.701,E2 -13535.701} C_VEL
LIN {X 0,Y 354.813,Z 168.289,A -85,B 0,C 180,E1 -13539.425,E2 -13539.425} C_VEL
LIN {X 0,Y 354.779,Z 168.29,A -85,B 0,C 180,E1 -13542.869,E2 -13542.869} C_VEL
LIN {X 0,Y 354.773,Z 168.292,A -85,B 0,C 180,E1 -13546.108,E2 -13546.108} C_VEL
LIN {X 0,Y 354.779,Z 168.294,A -85,B 0,C 180,E1 -13549.181,E2 -13549.181} C_VEL
LIN {X 0,Y 354.799,Z 168.287,A -85,B 0,C 180,E1 -13552.404,E2 -13552.404} C_VEL
LIN {X 0,Y 354.805,Z 168.29,A -85,B 0,C 180,E1 -13554.943,E2 -13554.943} C_VEL
LIN {X 0,Y 354.787,Z 168.29,A -85,B 0,C 180,E1 -13558.407,E2 -13558.407} C_VEL
LIN {X 0,Y 354.849,Z 168.282,A -85,B 0,C 180,E1 -13561.621,E2 -13561.621} C_VEL
LIN {X 0,Y 354.894,Z 168.276,A -85,B 0,C 180,E1 -13564.175,E2 -13564.175} C_VEL
